C03670=1113.021,-63.508,-48.459,179.722,5.253,148.994
C03671=1113.016,-63.258,-48.470,179.723,5.257,148.995
C03672=1113.010,-63.008,-48.481,179.723,5.262,148.995
C03673=1113.006,-62.759,-48.493,179.724,5.268,148.997
C03674=1113.001,-62.509,-48.504,179.724,5.273,148.998
C03675=1112.995,-62.259,-48.516,179.724,5.278,148.998
C03676=1112.990,-62.010,-48.526,179.725,5.283,148.999
C03677=1112.985,-61.760,-48.537,179.725,5.288,149.001
C03678=1112.980,-61.510,-48.549,179.726,5.293,149.001
C03679=1112.975,-61.260,-48.560,179.726,5.298,149.002
C03680=1112.969,-61.011,-48.572,179.727,5.303,149.003
C03681=1112.964,-60.761,-48.583,179.727,5.308,149.004
C03682=1112.959,-60.511,-48.594,179.727,5.313,149.005
C03683=1112.954,-60.261,-48.606,179.728,5.319,149.006
C03684=1112.949,-60.013,-48.617,179.729,5.324,149.007
C03685=1112.944,-59.798,-48.627,179.728,5.327,149.008
C03686=1112.940,-59.583,-48.637,179.728,5.331,149.009
C03687=1112.936,-59.368,-48.647,179.728,5.335,149.010
C03688=1112.930,-59.153,-48.656,179.728,5.339,149.011
C03689=1112.926,-58.938,-48.666,179.728,5.343,149.012
C03690=1112.922,-58.723,-48.676,179.728,5.348,149.013
C03691=1112.917,-58.509,-48.686,179.728,5.352,149.014
C03692=1112.913,-58.294,-48.696,179.728,5.356,149.015
C03693=1112.907,-58.044,-48.707,179.727,5.360,149.016
C03694=1112.902,-57.795,-48.718,179.727,5.365,149.017
C03695=1112.897,-57.545,-48.730,179.728,5.370,149.018
C03696=1112.892,-57.295,-48.742,179.727,5.374,149.019
C03697=1112.887,-57.045,-48.753,179.727,5.379,149.020
C03698=1112.882,-56.796,-48.765,179.727,5.384,149.021
C03699=1112.876,-56.546,-48.776,179.727,5.388,149.022
C03700=1112.871,-56.297,-48.788,179.727,5.393,149.023
C03701=1112.866,-56.047,-48.799,179.726,5.397,149.024
C03702=1112.861,-55.797,-48.811,179.726,5.403,149.025
C03703=1112.856,-55.547,-48.823,179.727,5.407,149.026
C03704=1112.851,-55.298,-48.834,179.726,5.412,149.027
C03705=1112.845,-55.048,-48.845,179.726,5.417,149.028
C03706=1112.840,-54.799,-48.857,179.726,5.421,149.029
C03707=1112.835,-54.549,-48.869,179.726,5.426,149.031
C03708=1112.829,-54.299,-48.881,179.726,5.431,149.032
C03709=1112.825,-54.049,-48.892,179.725,5.435,149.033
C03710=1112.819,-53.799,-48.904,179.725,5.440,149.034
C03711=1112.814,-53.549,-48.916,179.725,5.445,149.035
C03712=1112.809,-53.301,-48.927,179.725,5.449,149.036
C03713=1112.803,-53.051,-48.938,179.725,5.454,149.037
C03714=1112.799,-52.801,-48.950,179.724,5.459,149.038
C03715=1112.793,-52.551,-48.962,179.725,5.463,149.039
C03716=1112.788,-52.302,-48.974,179.725,5.468,149.040
C03717=1112.783,-52.052,-48.985,179.724,5.473,149.041
C03718=1112.778,-51.802,-48.997,179.724,5.478,149.042
C03719=1112.772,-51.552,-49.009,179.724,5.483,149.043
C03720=1112.767,-51.303,-49.020,179.724,5.487,149.045
C03721=1112.762,-51.053,-49.032,179.724,5.492,149.046
C03722=1112.756,-50.803,-49.044,179.723,5.496,149.047
C03723=1112.752,-50.554,-49.055,179.723,5.501,149.048
C03724=1112.746,-50.305,-49.068,179.724,5.506,149.049
C03725=1112.741,-50.055,-49.080,179.723,5.510,149.050
C03726=1112.736,-49.805,-49.091,179.723,5.515,149.051
C03727=1112.731,-49.555,-49.103,179.723,5.521,149.052
C03728=1112.725,-49.305,-49.115,179.723,5.524,149.053
C03729=1112.721,-49.056,-49.127,179.723,5.530,149.054
C03730=1112.716,-48.806,-49.139,179.722,5.534,149.055
C03731=1112.710,-48.556,-49.151,179.722,5.539,149.056
C03732=1112.705,-48.307,-49.161,179.722,5.544,149.057
C03733=1112.699,-48.057,-49.173,179.722,5.548,149.059
C03734=1112.694,-47.808,-49.186,179.722,5.553,149.060
C03735=1112.689,-47.558,-49.198,179.721,5.557,149.061
C03736=1112.684,-47.308,-49.209,179.721,5.562,149.062
C03737=1112.679,-47.059,-49.221,179.721,5.567,149.063
C03738=1112.674,-46.809,-49.234,179.721,5.571,149.064
C03739=1112.668,-46.559,-49.245,179.721,5.577,149.065
C03740=1112.664,-46.310,-49.257,179.721,5.582,149.066
C03741=1112.659,-46.095,-49.268,179.721,5.586,149.067
C03742=1112.654,-45.880,-49.278,179.721,5.590,149.068
C03743=1112.650,-45.665,-49.288,179.720,5.594,149.069
C03744=1112.646,-45.450,-49.298,179.720,5.597,149.070
C03745=1112.642,-45.236,-49.309,179.720,5.601,149.071
C03746=1112.637,-45.021,-49.319,179.720,5.605,149.072
C03747=1112.632,-44.807,-49.329,179.720,5.609,149.073
C03748=1112.628,-44.593,-49.340,179.720,5.613,149.074
C03749=1112.622,-44.343,-49.352,179.719,5.618,149.075
C03750=1112.617,-44.093,-49.364,179.719,5.623,149.076
C03751=1112.612,-43.843,-49.376,179.719,5.627,149.077
C03752=1112.607,-43.594,-49.387,179.719,5.633,149.078
C03753=1112.602,-43.344,-49.399,179.718,5.637,149.079
C03754=1112.596,-43.095,-49.412,179.718,5.642,149.080
C03755=1112.591,-42.845,-49.424,179.719,5.647,149.081
C03756=1112.587,-42.595,-49.437,179.719,5.652,149.082
C03757=1112.582,-42.345,-49.448,179.720,5.657,149.083
C03758=1112.576,-42.095,-49.460,179.721,5.663,149.084
C03759=1112.571,-41.846,-49.473,179.722,5.667,149.085
C03760=1112.566,-41.596,-49.484,179.723,5.673,149.086
C03761=1112.561,-41.347,-49.497,179.723,5.678,149.087
C03762=1112.555,-41.097,-49.509,179.724,5.683,149.087
C03763=1112.550,-40.847,-49.522,179.725,5.688,149.088
C03764=1112.545,-40.597,-49.533,179.726,5.693,149.089
C03765=1112.540,-40.348,-49.546,179.726,5.698,149.090
C03766=1112.534,-40.098,-49.558,179.727,5.703,149.091
C03767=1112.530,-39.849,-49.570,179.728,5.708,149.092
C03768=1112.524,-39.599,-49.582,179.729,5.713,149.093
C03769=1112.519,-39.350,-49.594,179.729,5.718,149.094
C03770=1112.514,-39.100,-49.606,179.730,5.723,149.094
C03771=1112.509,-38.851,-49.619,179.731,5.728,149.095
C03772=1112.504,-38.600,-49.631,179.732,5.732,149.096
C03773=1112.499,-38.351,-49.644,179.732,5.737,149.097
C03774=1112.494,-38.101,-49.656,179.732,5.742,149.098
C03775=1112.488,-37.851,-49.668,179.733,5.746,149.099
C03776=1112.483,-37.602,-49.681,179.734,5.752,149.100
C03777=1112.478,-37.352,-49.693,179.735,5.756,149.100
C03778=1112.473,-37.103,-49.705,179.735,5.761,149.101
C03779=1112.467,-36.853,-49.718,179.736,5.766,149.102
C03780=1112.462,-36.604,-49.730,179.736,5.771,149.103
C03781=1112.457,-36.353,-49.743,179.737,5.775,149.104
C03782=1112.452,-36.104,-49.755,179.738,5.780,149.105
C03783=1112.447,-35.854,-49.767,179.738,5.784,149.106
C03784=1112.442,-35.605,-49.780,179.738,5.788,149.106
C03785=1112.437,-35.356,-49.792,179.738,5.793,149.107
C03786=1112.430,-35.105,-49.805,179.739,5.797,149.108
C03787=1112.426,-34.855,-49.818,179.740,5.802,149.109
C03788=1112.421,-34.606,-49.830,179.740,5.807,149.110
C03789=1112.416,-34.357,-49.843,179.741,5.812,149.111
C03790=1112.410,-34.107,-49.855,179.740,5.816,149.112
C03791=1112.405,-33.857,-49.868,179.741,5.820,149.113
C03792=1112.401,-33.607,-49.881,179.742,5.825,149.113
C03793=1112.396,-33.358,-49.893,179.742,5.829,149.114
C03794=1112.390,-33.108,-49.905,179.742,5.833,149.115
C03795=1112.385,-32.859,-49.918,179.743,5.838,149.116
C03796=1112.380,-32.610,-49.930,179.743,5.843,149.117
C03797=1112.375,-32.395,-49.942,179.743,5.846,149.118
C03798=1112.371,-32.179,-49.952,179.743,5.850,149.118
C03799=1112.367,-31.965,-49.963,179.744,5.854,149.119
C03800=1112.363,-31.751,-49.974,179.743,5.858,149.120
C03801=1112.358,-31.536,-49.985,179.744,5.861,149.121
C03802=1112.353,-31.321,-49.995,179.744,5.865,149.121
C03803=1112.349,-31.107,-50.007,179.744,5.869,149.122
C03804=1112.345,-30.892,-50.017,179.744,5.872,149.123
C03805=1112.339,-30.643,-50.031,179.745,5.877,149.124
C03806=1112.334,-30.393,-50.043,179.745,5.881,149.125
C03807=1112.329,-30.143,-50.056,179.745,5.886,149.126
C03808=1112.324,-29.894,-50.069,179.745,5.890,149.127
C03809=1112.319,-29.644,-50.081,179.745,5.895,149.128
C03810=1112.314,-29.394,-50.094,179.745,5.899,149.129
C03811=1112.308,-29.145,-50.107,179.745,5.903,149.130
C03812=1112.303,-28.895,-50.119,179.745,5.907,149.130
C03813=1112.298,-28.646,-50.132,179.745,5.912,149.132
C03814=1112.293,-28.396,-50.145,179.745,5.916,149.133
C03815=1112.288,-28.147,-50.157,179.745,5.920,149.133
C03816=1112.282,-27.897,-50.171,179.745,5.925,149.134
C03817=1112.278,-27.647,-50.184,179.745,5.929,149.135
C03818=1112.273,-27.398,-50.196,179.745,5.933,149.136
C03819=1112.268,-27.148,-50.209,179.745,5.939,149.137
C03820=1112.262,-26.899,-50.222,179.744,5.942,149.138
C03821=1112.257,-26.649,-50.235,179.744,5.946,149.139
C03822=1112.252,-26.399,-50.248,179.744,5.952,149.140
C03823=1112.247,-26.150,-50.260,179.744,5.956,149.142
C03824=1112.242,-25.900,-50.274,179.744,5.960,149.142
C03825=1112.237,-25.650,-50.286,179.744,5.965,149.144
C03826=1112.232,-25.401,-50.299,179.744,5.970,149.145
C03827=1112.227,-25.151,-50.312,179.744,5.974,149.145
C03828=1112.221,-24.901,-50.325,179.745,5.979,149.146
C03829=1112.216,-24.652,-50.338,179.745,5.984,149.147
C03830=1112.211,-24.402,-50.351,179.746,5.989,149.148
C03831=1112.206,-24.152,-50.364,179.746,5.993,149.149
C03832=1112.200,-23.903,-50.377,179.747,5.998,149.150
C03833=1112.196,-23.653,-50.389,179.747,6.003,149.151
C03834=1112.190,-23.403,-50.403,179.748,6.007,149.152
C03835=1112.185,-23.154,-50.415,179.748,6.012,149.153
C03836=1112.180,-22.904,-50.428,179.749,6.017,149.154
C03837=1112.175,-22.655,-50.441,179.749,6.022,149.154
C03838=1112.170,-22.406,-50.455,179.750,6.026,149.155
C03839=1112.165,-22.156,-50.468,179.750,6.031,149.156
C03840=1112.159,-21.906,-50.481,179.751,6.036,149.157
C03841=1112.154,-21.657,-50.494,179.751,6.041,149.158
C03842=1112.149,-21.407,-50.507,179.752,6.045,149.159
C03843=1112.144,-21.157,-50.520,179.752,6.050,149.160
C03844=1112.140,-20.908,-50.533,179.753,6.055,149.161
C03845=1112.134,-20.658,-50.547,179.753,6.059,149.162
C03846=1112.129,-20.409,-50.559,179.754,6.064,149.163
C03847=1112.123,-20.159,-50.573,179.754,6.069,149.163
C03848=1112.118,-19.909,-50.585,179.754,6.073,149.164
C03849=1112.114,-19.660,-50.599,179.754,6.078,149.165
C03850=1112.108,-19.410,-50.612,179.755,6.082,149.166
C03851=1112.104,-19.160,-50.625,179.755,6.087,149.167
C03852=1112.098,-18.911,-50.638,179.756,6.092,149.168
C03853=1112.093,-18.697,-50.650,179.757,6.096,149.169
C03854=1112.089,-18.482,-50.661,179.757,6.100,149.169
C03855=1112.085,-18.267,-50.673,179.757,6.104,149.170
C03856=1112.080,-18.053,-50.684,179.758,6.108,149.171
C03857=1112.076,-17.838,-50.695,179.758,6.111,149.171
C03858=1112.072,-17.624,-50.706,179.759,6.116,149.172
C03859=1112.068,-17.409,-50.719,179.759,6.120,149.173
C03860=1112.063,-17.195,-50.730,179.760,6.123,149.174
C03861=1112.058,-16.945,-50.742,179.760,6.128,149.175
C03862=1112.053,-16.696,-50.757,179.761,6.133,149.176
C03863=1112.048,-16.446,-50.769,179.761,6.137,149.176
C03864=1112.042,-16.196,-50.783,179.762,6.142,149.177
C03865=1112.038,-15.947,-50.796,179.763,6.147,149.178
C03866=1112.032,-15.697,-50.810,179.763,6.151,149.179
C03867=1112.027,-15.448,-50.822,179.764,6.156,149.180
C03868=1112.022,-15.198,-50.837,179.764,6.161,149.181
C03869=1112.016,-14.948,-50.850,179.765,6.165,149.182
C03870=1112.012,-14.699,-50.864,179.765,6.170,149.182
C03871=1112.006,-14.449,-50.877,179.766,6.175,149.183
C03872=1112.002,-14.199,-50.890,179.767,6.179,149.184
C03873=1111.996,-13.950,-50.904,179.766,6.183,149.185
C03874=1111.992,-13.700,-50.917,179.767,6.188,149.186
C03875=1111.986,-13.451,-50.930,179.767,6.193,149.187
C03876=1111.981,-13.201,-50.944,179.768,6.197,149.187
C03877=1111.976,-12.952,-50.957,179.769,6.202,149.188
C03878=1111.971,-12.702,-50.971,179.769,6.206,149.189
C03879=1111.966,-12.453,-50.984,179.770,6.211,149.190
C03880=1111.961,-12.203,-50.998,179.771,6.215,149.191
C03881=1111.956,-11.953,-51.012,179.771,6.220,149.192
C03882=1111.951,-11.704,-51.025,179.772,6.225,149.193
C03883=1111.946,-11.454,-51.039,179.772,6.230,149.193
C03884=1111.940,-11.204,-51.052,179.773,6.233,149.194
C03885=1111.936,-10.955,-51.066,179.773,6.238,149.195
C03886=1111.930,-10.706,-51.080,179.774,6.243,149.196
C03887=1111.925,-10.456,-51.093,179.774,6.247,149.197
C03888=1111.921,-10.206,-51.107,179.775,6.252,149.197
C03889=1111.915,-9.957,-51.120,179.776,6.256,149.198
C03890=1111.910,-9.707,-51.134,179.776,6.261,149.199
C03891=1111.905,-9.458,-51.148,179.777,6.266,149.200
C03892=1111.900,-9.208,-51.161,179.778,6.270,149.201
C03893=1111.895,-8.958,-51.176,179.778,6.275,149.202
C03894=1111.890,-8.709,-51.188,179.778,6.279,149.203
C03895=1111.885,-8.459,-51.202,179.779,6.284,149.203
C03896=1111.880,-8.209,-51.217,179.780,6.288,149.204
C03897=1111.874,-7.960,-51.230,179.780,6.293,149.205
C03898=1111.870,-7.710,-51.244,179.781,6.297,149.206
C03899=1111.864,-7.461,-51.258,179.782,6.302,149.207
C03900=1111.859,-7.212,-51.272,179.782,6.306,149.207
C03901=1111.854,-6.961,-51.285,179.783,6.311,149.208
C03902=1111.849,-6.713,-51.299,179.783,6.316,149.209
C03903=1111.844,-6.463,-51.313,179.784,6.320,149.210
C03904=1111.839,-6.213,-51.327,179.784,6.324,149.211
C03905=1111.833,-5.964,-51.340,179.785,6.329,149.212
C03906=1111.829,-5.714,-51.354,179.786,6.333,149.212
C03907=1111.824,-5.464,-51.368,179.786,6.338,149.213
C03908=1111.818,-5.215,-51.382,179.787,6.343,149.214
C03909=1111.814,-5.000,-51.394,179.787,6.346,149.215
C03910=1111.810,-4.786,-51.406,179.788,6.350,149.215
C03911=1111.806,-4.571,-51.418,179.788,6.354,149.216
C03912=1111.801,-4.357,-51.430,179.788,6.358,149.217
C03913=1111.797,-4.143,-51.442,179.789,6.362,149.218
C03914=1111.793,-3.928,-51.453,179.790,6.366,149.218
C03915=1111.788,-3.714,-51.466,179.790,6.369,149.219
C03916=1111.784,-3.499,-51.478,179.791,6.374,149.220
C03917=1111.779,-3.250,-51.492,179.792,6.378,149.221
C03918=1111.774,-3.000,-51.505,179.792,6.383,149.222
C03919=1111.769,-2.750,-51.520,179.793,6.387,149.222
C03920=1111.763,-2.501,-51.534,179.793,6.391,149.223
C03921=1111.758,-2.252,-51.548,179.794,6.396,149.224
C03922=1111.753,-2.002,-51.562,179.794,6.401,149.225
C03923=1111.748,-1.752,-51.576,179.795,6.405,149.226
C03924=1111.743,-1.503,-51.590,179.796,6.410,149.226
C03925=1111.738,-1.253,-51.605,179.796,6.415,149.227
C03926=1111.733,-1.004,-51.618,179.797,6.419,149.228
C03927=1111.729,-0.754,-51.633,179.798,6.424,149.229
C03928=1111.723,-0.505,-51.646,179.798,6.428,149.230
C03929=1111.718,-0.256,-51.661,179.798,6.432,149.231
C03930=1111.713,-0.006,-51.675,179.799,6.437,149.231
C03931=1111.708,0.244,-51.689,179.800,6.441,149.232
C03932=1111.702,0.493,-51.702,179.800,6.446,149.233
C03933=1111.697,0.743,-51.717,179.801,6.450,149.234
C03934=1111.692,0.993,-51.731,179.802,6.455,149.235
C03935=1111.688,1.242,-51.746,179.802,6.460,149.236
C03936=1111.683,1.492,-51.760,179.803,6.464,149.236
C03937=1111.677,1.741,-51.774,179.804,6.469,149.237
C03938=1111.672,1.990,-51.788,179.804,6.474,149.238
C03939=1111.667,2.240,-51.803,179.804,6.477,149.239
C03940=1111.662,2.490,-51.817,179.805,6.482,149.240
C03941=1111.657,2.740,-51.831,179.806,6.486,149.240
C03942=1111.652,2.989,-51.845,179.806,6.491,149.241
C03943=1111.647,3.238,-51.860,179.807,6.496,149.242
C03944=1111.642,3.488,-51.874,179.807,6.501,149.243
C03945=1111.637,3.738,-51.888,179.808,6.505,149.244
C03946=1111.632,3.987,-51.902,179.809,6.510,149.245
C03947=1111.627,4.237,-51.917,179.810,6.514,149.245
C03948=1111.622,4.486,-51.932,179.810,6.519,149.246
C03949=1111.617,4.735,-51.946,179.811,6.523,149.247
C03950=1111.611,4.985,-51.960,179.812,6.528,149.248
C03951=1111.606,5.235,-51.975,179.812,6.533,149.249
C03952=1111.601,5.485,-51.989,179.812,6.537,149.250
C03953=1111.596,5.734,-52.003,179.813,6.541,149.251
C03954=1111.592,5.983,-52.018,179.814,6.546,149.251
C03955=1111.587,6.233,-52.033,179.814,6.551,149.252
C03956=1111.581,6.482,-52.046,179.815,6.555,149.253
C03957=1111.576,6.732,-52.061,179.815,6.560,149.254
C03958=1111.572,6.981,-52.076,179.816,6.565,149.255
C03959=1111.566,7.231,-52.091,179.817,6.569,149.255
C03960=1111.561,7.481,-52.105,179.817,6.574,149.256
C03961=1111.556,7.730,-52.119,179.818,6.578,149.257
C03962=1111.551,7.979,-52.134,179.818,6.583,149.258
C03963=1111.546,8.229,-52.148,179.819,6.588,149.259
C03964=1111.541,8.479,-52.163,179.820,6.593,149.260
C03965=1111.536,8.693,-52.175,179.820,6.596,149.261
C03966=1111.532,8.908,-52.188,179.820,6.600,149.261
C03967=1111.528,9.121,-52.200,179.821,6.604,149.262
C03968=1111.524,9.336,-52.213,179.821,6.608,149.263
C03969=1111.520,9.551,-52.226,179.822,6.611,149.263
C03970=1111.515,9.765,-52.238,179.822,6.616,149.264
C03971=1111.511,9.980,-52.251,179.823,6.620,149.265
C03972=1111.506,10.193,-52.263,179.823,6.623,149.266
C03973=1111.501,10.443,-52.278,179.824,6.628,149.267
C03974=1111.496,10.693,-52.293,179.824,6.633,149.267
C03975=1111.491,10.942,-52.307,179.825,6.637,149.268
C03976=1111.486,11.191,-52.322,179.826,6.642,149.269
C03977=1111.481,11.441,-52.336,179.826,6.646,149.270
C03978=1111.476,11.691,-52.352,179.826,6.650,149.271
C03979=1111.471,11.940,-52.366,179.827,6.655,149.272
C03980=1111.466,12.189,-52.381,179.827,6.660,149.272
C03981=1111.461,12.439,-52.395,179.828,6.664,149.273
C03982=1111.456,12.689,-52.410,179.829,6.669,149.274
C03983=1111.451,12.938,-52.425,179.830,6.673,149.275
C03984=1111.446,13.188,-52.440,179.829,6.677,149.276
C03985=1111.441,13.437,-52.455,179.830,6.682,149.276
C03986=1111.436,13.687,-52.469,179.831,6.686,149.277
C03987=1111.431,13.936,-52.484,179.832,6.691,149.278
C03988=1111.425,14.186,-52.499,179.833,6.695,149.279
C03989=1111.421,14.435,-52.514,179.833,6.700,149.280
C03990=1111.416,14.685,-52.529,179.833,6.704,149.281
C03991=1111.410,14.934,-52.544,179.834,6.709,149.282
C03992=1111.405,15.184,-52.558,179.835,6.713,149.282
C03993=1111.401,15.433,-52.573,179.835,6.718,149.283
C03994=1111.395,15.682,-52.589,179.836,6.722,149.284
C03995=1111.390,15.932,-52.603,179.837,6.727,149.285
C03996=1111.386,16.181,-52.618,179.837,6.731,149.285
C03997=1111.380,16.431,-52.633,179.838,6.735,149.286
C03998=1111.376,16.681,-52.649,179.838,6.740,149.287
C03999=1111.371,16.930,-52.664,179.839,6.744,149.288
C04000=1111.366,17.180,-52.678,179.840,6.749,149.289
C04001=1111.361,17.429,-52.693,179.841,6.753,149.289
C04002=1111.355,17.679,-52.708,179.841,6.757,149.290
C04003=1111.351,17.928,-52.723,179.842,6.762,149.291
C04004=1111.345,18.178,-52.739,179.843,6.766,149.292
C04005=1111.340,18.428,-52.753,179.843,6.771,149.293
C04006=1111.336,18.677,-52.768,179.844,6.775,149.293
C04007=1111.330,18.926,-52.784,179.844,6.779,149.294
C04008=1111.326,19.175,-52.799,179.845,6.784,149.295
C04009=1111.320,19.425,-52.814,179.846,6.788,149.296
C04010=1111.316,19.675,-52.829,179.846,6.793,149.296
C04011=1111.310,19.924,-52.844,179.847,6.797,149.297
C04012=1111.306,20.174,-52.859,179.848,6.802,149.298
C04013=1111.300,20.423,-52.874,179.848,6.805,149.299
C04014=1111.296,20.673,-52.889,179.849,6.809,149.299
C04015=1111.290,20.922,-52.905,179.850,6.814,149.300
C04016=1111.285,21.172,-52.919,179.851,6.818,149.301
C04017=1111.280,21.422,-52.935,179.852,6.823,149.302
C04018=1111.276,21.671,-52.950,179.852,6.827,149.302
C04019=1111.270,21.920,-52.966,179.853,6.831,149.303
C04020=1111.266,22.169,-52.981,179.854,6.836,149.304
C04021=1111.261,22.384,-52.994,179.854,6.839,149.305
C04022=1111.256,22.598,-53.007,179.855,6.844,149.305
C04023=1111.252,22.813,-53.019,179.856,6.847,149.306
C04024=1111.248,23.027,-53.033,179.856,6.851,149.307
C04025=1111.244,23.241,-53.046,179.856,6.854,149.307
C04026=1111.239,23.455,-53.059,179.857,6.858,149.308
C04027=1111.235,23.669,-53.073,179.858,6.862,149.308
C04028=1111.231,23.883,-53.086,179.859,6.865,149.309
C04029=1111.226,24.133,-53.101,179.859,6.870,149.310
C04030=1111.220,24.383,-53.116,179.860,6.874,149.311
C04031=1111.216,24.633,-53.132,179.861,6.878,149.311
C04032=1111.211,24.882,-53.147,179.861,6.882,149.312
C04033=1111.206,25.131,-53.162,179.863,6.887,149.313
C04034=1111.201,25.381,-53.178,179.864,6.891,149.313
C04035=1111.195,25.630,-53.193,179.864,6.896,149.314
C04036=1111.191,25.880,-53.209,179.865,6.900,149.315
C04037=1111.186,26.129,-53.224,179.866,6.903,149.316
C04038=1111.181,26.378,-53.239,179.866,6.908,149.316
C04039=1111.176,26.628,-53.255,179.867,6.912,149.317
C04040=1111.171,26.878,-53.271,179.868,6.917,149.318
C04041=1111.167,27.127,-53.286,179.869,6.921,149.318
C04042=1111.161,27.376,-53.301,179.869,6.925,149.319
C04043=1111.156,27.626,-53.317,179.870,6.929,149.320
C04044=1111.151,27.876,-53.333,179.871,6.934,149.321
C04045=1111.146,28.125,-53.348,179.872,6.938,149.321
C04046=1111.141,28.374,-53.363,179.874,6.942,149.322
C04047=1111.136,28.624,-53.379,179.874,6.946,149.323
C04048=1111.132,28.873,-53.394,179.875,6.950,149.323
C04049=1111.126,29.123,-53.410,179.876,6.955,149.324
C04050=1111.121,29.372,-53.426,179.877,6.959,149.325
C04051=1111.116,29.621,-53.441,179.877,6.963,149.325
C04052=1111.111,29.871,-53.457,179.878,6.967,149.326
C04053=1111.106,30.120,-53.473,179.879,6.972,149.327
C04054=1111.101,30.370,-53.488,179.880,6.976,149.328
C04055=1111.097,30.619,-53.504,179.881,6.980,149.328
C04056=1111.091,30.869,-53.519,179.881,6.984,149.329
C04057=1111.086,31.118,-53.535,179.882,6.988,149.330
C04058=1111.081,31.368,-53.551,179.883,6.993,149.330
C04059=1111.076,31.618,-53.567,179.884,6.997,149.331
C04060=1111.072,31.866,-53.582,179.885,7.001,149.332
C04061=1111.067,32.116,-53.598,179.886,7.005,149.332
C04062=1111.061,32.366,-53.614,179.887,7.009,149.333
C04063=1111.056,32.615,-53.629,179.888,7.014,149.334
C04064=1111.051,32.865,-53.645,179.889,7.018,149.334
C04065=1111.047,33.114,-53.661,179.890,7.022,149.335
C04066=1111.041,33.363,-53.677,179.890,7.026,149.336
C04067=1111.037,33.613,-53.693,179.891,7.030,149.336
C04068=1111.031,33.863,-53.708,179.892,7.034,149.337
C04069=1111.026,34.111,-53.724,179.893,7.039,149.338
C04070=1111.021,34.362,-53.740,179.894,7.043,149.338
C04071=1111.016,34.611,-53.756,179.894,7.047,149.339
C04072=1111.012,34.860,-53.772,179.896,7.051,149.340
C04073=1111.007,35.109,-53.788,179.897,7.055,149.340
C04074=1111.002,35.359,-53.803,179.898,7.060,149.341
C04075=1110.997,35.608,-53.820,179.898,7.063,149.342
C04076=1110.992,35.858,-53.836,179.899,7.068,149.342
C04077=1110.987,36.072,-53.849,179.900,7.071,149.343
C04078=1110.983,36.286,-53.863,179.901,7.075,149.344
C04079=1110.979,36.501,-53.877,179.902,7.078,149.344
C04080=1110.974,36.715,-53.890,179.903,7.082,149.345
C04081=1110.970,36.929,-53.904,179.904,7.086,149.345
C04082=1110.966,37.144,-53.918,179.905,7.089,149.346
C04083=1110.962,37.357,-53.932,179.905,7.093,149.346
C04084=1110.957,37.571,-53.946,179.906,7.096,149.347
C04085=1110.953,37.821,-53.961,179.907,7.100,149.347
C04086=1110.948,38.070,-53.977,179.908,7.104,149.348
C04087=1110.943,38.320,-53.993,179.909,7.109,149.349
C04088=1110.938,38.569,-54.009,179.910,7.112,149.349
C04089=1110.933,38.819,-54.025,179.911,7.116,149.350
C04090=1110.928,39.068,-54.041,179.912,7.121,149.351
C04091=1110.923,39.317,-54.058,179.913,7.125,149.351
C04092=1110.918,39.567,-54.073,179.914,7.129,149.352
C04093=1110.913,39.816,-54.090,179.915,7.133,149.352
C04094=1110.908,40.066,-54.105,179.916,7.137,149.353
C04095=1110.903,40.315,-54.122,179.917,7.141,149.354
C04096=1110.898,40.565,-54.138,179.918,7.145,149.354
C04097=1110.892,40.814,-54.155,179.919,7.150,149.355
C04098=1110.888,41.064,-54.171,179.919,7.153,149.356
C04099=1110.883,41.313,-54.187,179.921,7.158,149.356
C04100=1110.878,41.562,-54.204,179.922,7.161,149.357
C04101=1110.873,41.812,-54.219,179.923,7.166,149.357
C04102=1110.868,42.061,-54.236,179.924,7.169,149.358
C04103=1110.863,42.310,-54.251,179.925,7.174,149.359
C04104=1110.858,42.560,-54.268,179.926,7.178,149.359
C04105=1110.854,42.810,-54.284,179.927,7.182,149.360
C04106=1110.848,43.059,-54.300,179.928,7.186,149.361
C04107=1110.844,43.308,-54.317,179.929,7.190,149.361
C04108=1110.839,43.558,-54.333,179.930,7.194,149.362
C04109=1110.834,43.807,-54.349,179.931,7.198,149.362
C04110=1110.828,44.056,-54.366,179.932,7.203,149.363
C04111=1110.824,44.306,-54.382,179.934,7.206,149.364
C04112=1110.818,44.555,-54.398,179.934,7.210,149.364
C04113=1110.814,44.805,-54.415,179.935,7.214,149.365
C04114=1110.809,45.055,-54.431,179.936,7.219,149.366
C04115=1110.804,45.304,-54.447,179.937,7.223,149.366
C04116=1110.800,45.553,-54.464,179.939,7.227,149.367
C04117=1110.794,45.802,-54.481,179.939,7.230,149.367
C04118=1110.789,46.052,-54.497,179.940,7.235,149.368
C04119=1110.784,46.301,-54.513,179.942,7.239,149.369
C04120=1110.779,46.550,-54.530,179.943,7.243,149.369
C04121=1110.775,46.800,-54.547,179.944,7.247,149.370
C04122=1110.769,47.050,-54.563,179.945,7.251,149.370
C04123=1110.764,47.299,-54.579,179.946,7.255,149.371
C04124=1110.760,47.549,-54.596,179.947,7.259,149.371
C04125=1110.755,47.797,-54.612,179.948,7.263,149.372
C04126=1110.750,48.047,-54.629,179.949,7.267,149.373
C04127=1110.745,48.296,-54.646,179.950,7.271,149.373
C04128=1110.740,48.546,-54.662,179.951,7.275,149.374
C04129=1110.735,48.796,-54.679,179.952,7.279,149.374
C04130=1110.730,49.044,-54.695,179.954,7.283,149.375
C04131=1110.725,49.294,-54.712,179.955,7.287,149.376
C04132=1110.720,49.544,-54.729,179.956,7.291,149.376
C04133=1110.716,49.758,-54.742,179.957,7.295,149.377
C04134=1110.712,49.972,-54.757,179.958,7.298,149.377
C04135=1110.707,50.186,-54.772,179.959,7.301,149.378
C04136=1110.703,50.400,-54.786,179.959,7.305,149.378
C04137=1110.699,50.614,-54.800,179.961,7.308,149.379
C04138=1110.695,50.828,-54.814,179.962,7.312,149.379
C04139=1110.690,51.042,-54.829,179.962,7.315,149.380
C04140=1110.686,51.256,-54.843,179.963,7.318,149.380
C04141=1110.682,51.505,-54.860,179.964,7.323,149.381
C04142=1110.676,51.755,-54.877,179.966,7.326,149.381
C04143=1110.671,52.004,-54.893,179.967,7.331,149.382
C04144=1110.667,52.253,-54.910,179.969,7.335,149.382
C04145=1110.662,52.503,-54.927,179.970,7.339,149.383
C04146=1110.657,52.753,-54.944,179.970,7.342,149.384
C04147=1110.652,53.001,-54.960,179.972,7.346,149.384
C04148=1110.647,53.251,-54.978,179.973,7.351,149.385
C04149=1110.642,53.501,-54.994,179.974,7.355,149.385
C04150=1110.637,53.750,-55.011,179.975,7.359,149.386
C04151=1110.632,53.999,-55.028,179.976,7.362,149.386
C04152=1110.628,54.249,-55.045,179.978,7.366,149.387
C04153=1110.622,54.498,-55.062,179.979,7.371,149.387
C04154=1110.617,54.747,-55.078,179.980,7.375,149.388
C04155=1110.612,54.997,-55.095,179.981,7.379,149.389
C04156=1110.608,55.247,-55.112,179.983,7.383,149.389
C04157=1110.603,55.496,-55.130,179.983,7.386,149.390
C04158=1110.598,55.745,-55.146,179.985,7.390,149.390
C04159=1110.592,55.994,-55.164,179.986,7.394,149.391
C04160=1110.588,56.244,-55.180,179.987,7.399,149.391
C04161=1110.583,56.494,-55.197,179.989,7.403,149.392
C04162=1110.578,56.743,-55.214,179.989,7.406,149.392
C04163=1110.573,56.992,-55.230,179.991,7.410,149.393
C04164=1110.568,57.241,-55.248,179.992,7.414,149.394
C04165=1110.563,57.491,-55.266,179.993,7.418,149.394
C04166=1110.559,57.740,-55.282,179.994,7.423,149.395
C04167=1110.553,57.990,-55.300,179.996,7.426,149.395
C04168=1110.549,58.238,-55.317,179.996,7.430,149.396
C04169=1110.543,58.488,-55.334,179.998,7.434,149.396
C04170=1110.539,58.738,-55.351,179.999,7.438,149.397
C04171=1110.534,58.987,-55.368,-179.999,7.442,149.397
C04172=1110.529,59.236,-55.385,-179.998,7.446,149.398
C04173=1110.524,59.486,-55.403,-179.997,7.450,149.398
C04174=1110.519,59.735,-55.419,-179.996,7.454,149.399
C04175=1110.514,59.984,-55.437,-179.995,7.458,149.399
C04176=1110.509,60.234,-55.454,-179.994,7.462,149.400
C04177=1110.505,60.483,-55.471,-179.992,7.466,149.400
C04178=1110.500,60.732,-55.489,-179.990,7.470,149.401
C04179=1110.495,60.982,-55.505,-179.989,7.474,149.402
C04180=1110.490,61.232,-55.523,-179.988,7.477,149.402
C04181=1110.484,61.480,-55.540,-179.987,7.482,149.403
C04182=1110.480,61.730,-55.557,-179.986,7.485,149.403
C04183=1110.475,61.979,-55.575,-179.985,7.490,149.404
C04184=1110.471,62.228,-55.592,-179.983,7.494,149.404
C04185=1110.465,62.478,-55.609,-179.982,7.498,149.405
C04186=1110.460,62.727,-55.627,-179.981,7.501,149.405
C04187=1110.456,62.977,-55.643,-179.979,7.505,149.406
C04188=1110.451,63.226,-55.661,-179.978,7.509,149.406
C04189=1110.446,63.440,-55.676,-179.977,7.513,149.407
C04190=1110.442,63.654,-55.691,-179.976,7.516,149.407
C04191=1110.438,63.868,-55.706,-179.975,7.519,149.408
C04192=1110.434,64.082,-55.721,-179.974,7.522,149.408
C04193=1110.429,64.296,-55.736,-179.972,7.526,149.409
C04194=1110.426,64.510,-55.750,-179.971,7.530,149.409
C04195=1110.421,64.725,-55.766,-179.971,7.533,149.409
C04196=1110.418,64.938,-55.781,-179.969,7.537,149.410
C04197=1110.412,65.187,-55.798,-179.968,7.541,149.410
C04198=1110.408,65.437,-55.816,-179.967,7.544,149.411
C04199=1110.402,65.686,-55.833,-179.966,7.548,149.412
C04200=1110.398,65.935,-55.851,-179.964,7.552,149.412
C04201=1110.393,66.185,-55.868,-179.963,7.556,149.412
C04202=1110.388,66.434,-55.886,-179.962,7.560,149.413
C04203=1110.383,66.683,-55.904,-179.960,7.564,149.414
C04204=1110.379,66.933,-55.920,-179.959,7.569,149.414
C04205=1110.374,67.182,-55.938,-179.958,7.572,149.415
C04206=1110.369,67.432,-55.956,-179.956,7.576,149.415
C04207=1110.364,67.681,-55.974,-179.955,7.580,149.416
C04208=1110.359,67.930,-55.992,-179.954,7.584,149.416
C04209=1110.354,68.180,-56.008,-179.952,7.588,149.417
C04210=1110.349,68.429,-56.026,-179.951,7.592,149.417
C04211=1110.344,68.678,-56.044,-179.949,7.596,149.418
C04212=1110.339,68.928,-56.062,-179.948,7.600,149.418
C04213=1110.334,69.177,-56.080,-179.947,7.603,149.419
C04214=1110.329,69.426,-56.098,-179.946,7.607,149.419
C04215=1110.325,69.675,-56.115,-179.944,7.611,149.420
C04216=1110.320,69.925,-56.132,-179.943,7.615,149.420
C04217=1110.315,70.174,-56.150,-179.942,7.619,149.421
C04218=1110.310,70.423,-56.168,-179.940,7.623,149.421
C04219=1110.305,70.672,-56.186,-179.939,7.627,149.422
C04220=1110.300,70.922,-56.203,-179.937,7.631,149.422
C04221=1110.295,71.171,-56.221,-179.936,7.635,149.423
C04222=1110.290,71.420,-56.239,-179.935,7.639,149.423
C04223=1110.286,71.669,-56.257,-179.934,7.643,149.424
C04224=1110.281,71.919,-56.275,-179.932,7.647,149.424
C04225=1110.276,72.168,-56.293,-179.931,7.651,149.425
C04226=1110.272,72.418,-56.310,-179.929,7.655,149.425
C04227=1110.267,72.667,-56.328,-179.928,7.659,149.426
C04228=1110.262,72.917,-56.346,-179.927,7.663,149.426
C04229=1110.257,73.166,-56.364,-179.925,7.667,149.427
C04230=1110.252,73.415,-56.382,-179.924,7.671,149.427
C04231=1110.247,73.664,-56.400,-179.922,7.675,149.428
C04232=1110.242,73.913,-56.418,-179.921,7.678,149.428
C04233=1110.237,74.162,-56.436,-179.920,7.682,149.429
C04234=1110.232,74.412,-56.454,-179.918,7.686,149.429
C04235=1110.228,74.662,-56.472,-179.917,7.690,149.430
C04236=1110.223,74.911,-56.490,-179.916,7.694,149.430
C04237=1110.218,75.160,-56.508,-179.914,7.698,149.431
C04238=1110.213,75.410,-56.526,-179.912,7.702,149.431
C04239=1110.208,75.659,-56.544,-179.911,7.706,149.432
C04240=1110.203,75.908,-56.562,-179.910,7.710,149.432
C04241=1110.198,76.157,-56.580,-179.908,7.714,149.433
C04242=1110.194,76.407,-56.598,-179.907,7.718,149.433
C04243=1110.189,76.656,-56.616,-179.905,7.722,149.434
C04244=1110.184,76.905,-56.634,-179.904,7.726,149.434
C04245=1110.180,77.119,-56.650,-179.904,7.728,149.435
C04246=1110.176,77.333,-56.666,-179.903,7.731,149.435
C04247=1110.171,77.547,-56.681,-179.902,7.735,149.436
C04248=1110.167,77.761,-56.697,-179.901,7.738,149.436
C04249=1110.163,77.974,-56.713,-179.900,7.741,149.436
C04250=1110.159,78.189,-56.728,-179.899,7.744,149.437
C04251=1110.154,78.402,-56.744,-179.898,7.747,149.437
C04252=1110.150,78.617,-56.760,-179.898,7.751,149.438
C04253=1110.146,78.866,-56.778,-179.896,7.755,149.438
C04254=1110.141,79.115,-56.796,-179.896,7.758,149.439
C04255=1110.136,79.364,-56.814,-179.894,7.762,149.440
C04256=1110.131,79.614,-56.832,-179.894,7.766,149.440
C04257=1110.127,79.863,-56.850,-179.892,7.770,149.441
C04258=1110.122,80.112,-56.868,-179.891,7.773,149.441
C04259=1110.116,80.361,-56.887,-179.890,7.777,149.442
C04260=1110.112,80.611,-56.906,-179.889,7.781,149.442
C04261=1110.107,80.860,-56.924,-179.888,7.785,149.443
C04262=1110.102,81.109,-56.942,-179.887,7.788,149.443
C04263=1110.097,81.359,-56.960,-179.886,7.792,149.444
C04264=1110.093,81.608,-56.979,-179.885,7.795,149.444
C04265=1110.088,81.857,-56.997,-179.884,7.800,149.445
C04266=1110.083,82.107,-57.015,-179.883,7.803,149.446
C04267=1110.078,82.356,-57.033,-179.882,7.807,149.446
C04268=1110.074,82.605,-57.052,-179.880,7.811,149.447
C04269=1110.069,82.854,-57.070,-179.880,7.814,149.447
C04270=1110.063,83.104,-57.089,-179.878,7.818,149.448
C04271=1110.058,83.353,-57.107,-179.878,7.822,149.448
C04272=1110.054,83.602,-57.126,-179.876,7.826,149.449
C04273=1110.049,83.851,-57.144,-179.875,7.830,149.449
C04274=1110.044,84.101,-57.162,-179.874,7.833,149.450
C04275=1110.040,84.350,-57.182,-179.873,7.837,149.450
C04276=1110.035,84.599,-57.200,-179.871,7.841,149.451
C04277=1110.030,84.848,-57.218,-179.870,7.844,149.451
C04278=1110.025,85.098,-57.237,-179.869,7.849,149.452
C04279=1110.020,85.347,-57.255,-179.868,7.852,149.452
C04280=1110.015,85.596,-57.273,-179.867,7.856,149.453
C04281=1110.011,85.846,-57.293,-179.866,7.860,149.454
C04282=1110.006,86.095,-57.311,-179.865,7.863,149.454
C04283=1110.001,86.344,-57.329,-179.864,7.867,149.455
C04284=1109.996,86.594,-57.348,-179.862,7.871,149.455
C04285=1109.991,86.843,-57.366,-179.861,7.875,149.456
C04286=1109.986,87.091,-57.385,-179.860,7.879,149.456
C04287=1109.981,87.342,-57.404,-179.858,7.882,149.457
C04288=1109.977,87.590,-57.423,-179.858,7.886,149.457
C04289=1109.972,87.839,-57.441,-179.856,7.890,149.458
C04290=1109.967,88.089,-57.460,-179.855,7.894,149.458
C04291=1109.962,88.338,-57.478,-179.854,7.897,149.459
C04292=1109.957,88.587,-57.498,-179.852,7.901,149.459
C04293=1109.953,88.837,-57.516,-179.851,7.905,149.460
C04294=1109.948,89.085,-57.535,-179.850,7.909,149.460
C04295=1109.943,89.336,-57.554,-179.849,7.912,149.461
C04296=1109.938,89.584,-57.572,-179.847,7.916,149.461
C04297=1109.933,89.834,-57.591,-179.846,7.921,149.462
C04298=1109.929,90.083,-57.610,-179.844,7.924,149.462
C04299=1109.924,90.332,-57.628,-179.843,7.928,149.463
C04300=1109.919,90.582,-57.648,-179.842,7.931,149.463
C04301=1109.915,90.795,-57.663,-179.841,7.935,149.464
C04302=1109.911,91.009,-57.679,-179.840,7.938,149.464
C04303=1109.907,91.223,-57.695,-179.838,7.942,149.464
C04304=1109.902,91.437,-57.712,-179.837,7.945,149.465
C04305=1109.898,91.650,-57.729,-179.836,7.948,149.465
C04306=1109.894,91.865,-57.745,-179.835,7.951,149.466
C04307=1109.890,92.078,-57.760,-179.834,7.955,149.466
C04308=1109.886,92.292,-57.777,-179.833,7.958,149.467
C04309=1109.881,92.541,-57.796,-179.831,7.962,149.467
C04310=1109.877,92.791,-57.814,-179.830,7.965,149.467
C04311=1109.871,93.040,-57.834,-179.829,7.969,149.468
C04312=1109.867,93.289,-57.853,-179.827,7.973,149.468
C04313=1109.862,93.538,-57.871,-179.826,7.977,149.469
C04314=1109.858,93.788,-57.890,-179.824,7.981,149.469
C04315=1109.852,94.037,-57.909,-179.823,7.984,149.470
C04316=1109.848,94.286,-57.929,-179.822,7.988,149.470
C04317=1109.843,94.535,-57.947,-179.820,7.992,149.471
C04318=1109.838,94.785,-57.967,-179.819,7.996,149.471
C04319=1109.833,95.033,-57.985,-179.817,7.999,149.472
C04320=1109.828,95.283,-58.005,-179.816,8.003,149.472
C04321=1109.824,95.532,-58.023,-179.814,8.006,149.472
C04322=1109.819,95.782,-58.043,-179.813,8.011,149.473
C04323=1109.813,96.031,-58.062,-179.812,8.015,149.474
C04324=1109.809,96.280,-58.081,-179.810,8.019,149.474
C04325=1109.804,96.529,-58.100,-179.808,8.022,149.474
C04326=1109.800,96.778,-58.119,-179.807,8.026,149.475
C04327=1109.794,97.027,-58.138,-179.806,8.029,149.475
C04328=1109.790,97.277,-58.158,-179.804,8.033,149.476
C04329=1109.785,97.526,-58.176,-179.803,8.037,149.476
C04330=1109.780,97.775,-58.196,-179.801,8.041,149.477
C04331=1109.775,98.024,-58.215,-179.799,8.045,149.477
C04332=1109.771,98.273,-58.234,-179.798,8.049,149.477
C04333=1109.766,98.523,-58.254,-179.796,8.053,149.478
C04334=1109.761,98.772,-58.273,-179.795,8.055,149.478
C04335=1109.757,99.021,-58.292,-179.793,8.059,149.479
C04336=1109.752,99.270,-58.312,-179.792,8.063,149.479
C04337=1109.747,99.519,-58.331,-179.790,8.067,149.479
C04338=1109.742,99.768,-58.350,-179.788,8.071,149.480
C04339=1109.737,100.018,-58.369,-179.787,8.075,149.480
C04340=1109.732,100.268,-58.389,-179.785,8.079,149.481
C04341=1109.727,100.517,-58.408,-179.784,8.083,149.481
C04342=1109.723,100.765,-58.428,-179.782,8.086,149.481
C04343=1109.718,101.014,-58.447,-179.780,8.090,149.482
C04344=1109.713,101.264,-58.467,-179.779,8.093,149.482
C04345=1109.709,101.513,-58.486,-179.777,8.097,149.483
C04346=1109.704,101.762,-58.505,-179.776,8.101,149.483
C04347=1109.699,102.011,-58.525,-179.774,8.104,149.483
C04348=1109.695,102.261,-58.544,-179.772,8.108,149.484
C04349=1109.689,102.510,-58.564,-179.771,8.112,149.484
C04350=1109.685,102.759,-58.583,-179.769,8.116,149.485
C04351=1109.680,103.009,-58.602,-179.767,8.120,149.485
C04352=1109.675,103.257,-58.622,-179.765,8.123,149.485
C04353=1109.670,103.507,-58.641,-179.764,8.127,149.486
C04354=1109.666,103.756,-58.662,-179.762,8.131,149.486
C04355=1109.661,104.005,-58.681,-179.760,8.135,149.486
C04356=1109.657,104.254,-58.700,-179.758,8.139,149.487
C04357=1109.652,104.468,-58.717,-179.757,8.141,149.487
C04358=1109.648,104.682,-58.734,-179.755,8.145,149.487
C04359=1109.644,104.895,-58.751,-179.754,8.148,149.488
C04360=1109.640,105.109,-58.767,-179.752,8.151,149.488
C04361=1109.636,105.323,-58.784,-179.751,8.155,149.488
C04362=1109.631,105.537,-58.801,-179.749,8.157,149.489
C04363=1109.628,105.750,-58.818,-179.747,8.161,149.489
C04364=1109.623,105.965,-58.835,-179.746,8.164,149.489
C04365=1109.618,106.213,-58.855,-179.744,8.167,149.489
C04366=1109.614,106.462,-58.874,-179.743,8.171,149.490
C04367=1109.609,106.712,-58.894,-179.741,8.175,149.490
C04368=1109.605,106.961,-58.914,-179.739,8.179,149.491
C04369=1109.600,107.209,-58.933,-179.737,8.182,149.491
C04370=1109.595,107.459,-58.953,-179.735,8.186,149.491
C04371=1109.590,107.708,-58.973,-179.733,8.190,149.491
C04372=1109.586,107.958,-58.993,-179.731,8.193,149.492
C04373=1109.580,108.206,-59.012,-179.730,8.197,149.492
C04374=1109.576,108.455,-59.033,-179.728,8.200,149.492
C04375=1109.571,108.705,-59.052,-179.726,8.204,149.493
C04376=1109.566,108.955,-59.072,-179.724,8.208,149.493
C04377=1109.561,109.203,-59.092,-179.722,8.211,149.493
C04378=1109.557,109.452,-59.112,-179.720,8.215,149.494
C04379=1109.552,109.701,-59.132,-179.718,8.219,149.494
C04380=1109.548,109.951,-59.152,-179.716,8.222,149.494
C04381=1109.543,110.200,-59.172,-179.714,8.226,149.494
C04382=1109.538,110.449,-59.191,-179.713,8.230,149.495
C04383=1109.533,110.698,-59.212,-179.710,8.233,149.495
C04384=1109.529,110.947,-59.231,-179.708,8.237,149.495
C04385=1109.524,111.196,-59.252,-179.706,8.240,149.495
C04386=1109.519,111.446,-59.272,-179.705,8.244,149.496
C04387=1109.514,111.695,-59.292,-179.703,8.247,149.496
C04388=1109.509,111.944,-59.312,-179.702,8.251,149.497
C04389=1109.504,112.193,-59.332,-179.700,8.254,149.497
C04390=1109.500,112.442,-59.352,-179.698,8.258,149.497
C04391=1109.495,112.691,-59.372,-179.697,8.261,149.497
C04392=1109.490,112.941,-59.392,-179.695,8.264,149.498
C04393=1109.486,113.190,-59.412,-179.692,8.268,149.498
C04394=1109.482,113.439,-59.433,-179.691,8.272,149.498
C04395=1109.476,113.688,-59.452,-179.689,8.274,149.499
C04396=1109.471,113.937,-59.473,-179.687,8.278,149.499
C04397=1109.467,114.186,-59.493,-179.686,8.282,149.499
C04398=1109.462,114.435,-59.513,-179.684,8.284,149.499
C04399=1109.457,114.684,-59.533,-179.682,8.288,149.500
C04400=1109.452,114.934,-59.553,-179.681,8.292,149.500
C04401=1109.448,115.183,-59.574,-179.679,8.295,149.500
C04402=1109.443,115.432,-59.594,-179.677,8.298,149.501
C04403=1109.439,115.681,-59.615,-179.676,8.302,149.501
C04404=1109.433,115.930,-59.634,-179.673,8.305,149.501
C04405=1109.428,116.179,-59.655,-179.672,8.308,149.501
C04406=1109.424,116.428,-59.675,-179.670,8.312,149.502
C04407=1109.419,116.677,-59.696,-179.668,8.315,149.502
C04408=1109.415,116.927,-59.715,-179.666,8.319,149.502
C04409=1109.409,117.176,-59.736,-179.665,8.322,149.503
C04410=1109.405,117.425,-59.757,-179.663,8.326,149.503
C04411=1109.401,117.674,-59.777,-179.661,8.329,149.503
C04412=1109.396,117.923,-59.797,-179.660,8.332,149.503
C04413=1109.392,118.137,-59.815,-179.658,8.335,149.504
C04414=1109.388,118.350,-59.832,-179.656,8.338,149.504
C04415=1109.383,118.564,-59.850,-179.655,8.341,149.504
C04416=1109.379,118.778,-59.867,-179.654,8.344,149.505
C04417=1109.375,118.991,-59.885,-179.652,8.347,149.505
C04418=1109.372,119.205,-59.902,-179.651,8.349,149.505
C04419=1109.367,119.418,-59.919,-179.649,8.353,149.505
C04420=1109.363,119.632,-59.937,-179.647,8.355,149.505
C04421=1109.358,119.881,-59.958,-179.645,8.359,149.506
C04422=1109.353,120.130,-59.978,-179.644,8.362,149.506
C04423=1109.349,120.379,-59.998,-179.642,8.366,149.506
C04424=1109.344,120.629,-60.019,-179.640,8.369,149.507
C04425=1109.339,120.877,-60.040,-179.639,8.372,149.507
C04426=1109.335,121.126,-60.060,-179.637,8.376,149.507
C04427=1109.330,121.376,-60.081,-179.635,8.379,149.507
C04428=1109.325,121.625,-60.101,-179.634,8.382,149.508
C04429=1109.321,121.874,-60.122,-179.632,8.385,149.508
C04430=1109.316,122.123,-60.143,-179.630,8.389,149.508
C04431=1109.312,122.373,-60.164,-179.629,8.392,149.509
C04432=1109.307,122.622,-60.184,-179.627,8.395,149.509
C04433=1109.302,122.871,-60.205,-179.624,8.399,149.509
C04434=1109.298,123.120,-60.225,-179.623,8.402,149.510
C04435=1109.293,123.369,-60.246,-179.621,8.406,149.510
C04436=1109.288,123.618,-60.267,-179.619,8.409,149.510
C04437=1109.283,123.867,-60.288,-179.617,8.413,149.510
C04438=1109.279,124.116,-60.308,-179.616,8.416,149.511
C04439=1109.273,124.365,-60.329,-179.614,8.419,149.511
C04440=1109.269,124.614,-60.349,-179.612,8.423,149.511
C04441=1109.264,124.863,-60.371,-179.611,8.425,149.511
C04442=1109.260,125.112,-60.391,-179.609,8.429,149.512
C04443=1109.255,125.361,-60.412,-179.607,8.433,149.512
C04444=1109.251,125.611,-60.433,-179.606,8.435,149.512
C04445=1109.246,125.860,-60.454,-179.603,8.439,149.512
C04446=1109.241,126.109,-60.474,-179.602,8.443,149.513
C04447=1109.236,126.358,-60.495,-179.600,8.446,149.513
C04448=1109.232,126.607,-60.516,-179.598,8.449,149.513
C04449=1109.227,126.856,-60.537,-179.596,8.453,149.514
C04450=1109.222,127.105,-60.558,-179.595,8.455,149.514
C04451=1109.218,127.355,-60.579,-179.593,8.459,149.514
C04452=1109.213,127.604,-60.599,-179.591,8.463,149.514
C04453=1109.208,127.852,-60.621,-179.590,8.465,149.515
C04454=1109.204,128.101,-60.641,-179.588,8.469,149.515
C04455=1109.199,128.351,-60.662,-179.586,8.473,149.515
C04456=1109.194,128.599,-60.684,-179.585,8.475,149.516
C04457=1109.189,128.848,-60.705,-179.583,8.479,149.516
C04458=1109.185,129.098,-60.726,-179.580,8.482,149.516
C04459=1109.180,129.347,-60.747,-179.579,8.486,149.516
C04460=1109.176,129.596,-60.768,-179.577,8.489,149.517
C04461=1109.170,129.845,-60.789,-179.575,8.492,149.517
C04462=1109.166,130.094,-60.809,-179.573,8.496,149.517
C04463=1109.161,130.343,-60.831,-179.572,8.499,149.518
C04464=1109.156,130.593,-60.852,-179.570,8.503,149.518
C04465=1109.152,130.841,-60.873,-179.568,8.506,149.518
C04466=1109.147,131.090,-60.894,-179.567,8.509,149.518
C04467=1109.142,131.339,-60.915,-179.565,8.513,149.519
C04468=1109.138,131.588,-60.936,-179.563,8.516,149.519
C04469=1109.133,131.802,-60.955,-179.562,8.519,149.519
C04470=1109.130,132.016,-60.973,-179.560,8.522,149.519
C04471=1109.126,132.229,-60.991,-179.559,8.524,149.520
C04472=1109.122,132.442,-61.009,-179.557,8.527,149.520
C04473=1109.118,132.656,-61.028,-179.556,8.530,149.520
C04474=1109.113,132.870,-61.046,-179.554,8.534,149.521
C04475=1109.109,133.083,-61.064,-179.553,8.536,149.521
C04476=1109.105,133.296,-61.082,-179.551,8.539,149.521
C04477=1109.101,133.546,-61.104,-179.549,8.543,149.521
C04478=1109.096,133.795,-61.125,-179.548,8.545,149.521
C04479=1109.092,134.043,-61.146,-179.546,8.549,149.522
C04480=1109.087,134.292,-61.167,-179.544,8.553,149.522
C04481=1109.082,134.542,-61.189,-179.543,8.555,149.522
C04482=1109.077,134.791,-61.210,-179.541,8.559,149.523
C04483=1109.073,135.039,-61.231,-179.539,8.563,149.523
C04484=1109.069,135.289,-61.252,-179.537,8.565,149.523
C04485=1109.064,135.538,-61.274,-179.535,8.569,149.524
C04486=1109.058,135.787,-61.295,-179.534,8.573,149.524
C04487=1109.054,136.036,-61.317,-179.532,8.575,149.524
C04488=1109.050,136.285,-61.338,-179.530,8.579,149.524
C04489=1109.045,136.534,-61.359,-179.529,8.583,149.525
C04490=1109.040,136.783,-61.381,-179.527,8.586,149.525
C04491=1109.036,137.032,-61.403,-179.525,8.589,149.525
C04492=1109.031,137.281,-61.424,-179.523,8.593,149.526
C04493=1109.026,137.530,-61.445,-179.521,8.596,149.526
C04494=1109.022,137.779,-61.467,-179.520,8.599,149.526
C04495=1109.017,138.028,-61.488,-179.518,8.603,149.527
C04496=1109.012,138.277,-61.510,-179.516,8.606,149.527
C04497=1109.008,138.526,-61.532,-179.515,8.609,149.527
C04498=1109.003,138.775,-61.553,-179.513,8.613,149.528
C04499=1108.998,139.024,-61.574,-179.511,8.617,149.528
C04500=1108.994,139.274,-61.596,-179.509,8.620,149.528
C04501=1108.989,139.522,-61.618,-179.508,8.623,149.528
C04502=1108.984,139.772,-61.640,-179.506,8.627,149.529
C04503=1108.979,140.021,-61.661,-179.504,8.630,149.529
C04504=1108.975,140.269,-61.682,-179.503,8.633,149.529
C04505=1108.971,140.518,-61.704,-179.501,8.637,149.530
C04506=1108.966,140.767,-61.726,-179.499,8.641,149.530
C04507=1108.962,141.016,-61.748,-179.498,8.643,149.530
C04508=1108.957,141.266,-61.769,-179.496,8.647,149.531
C04509=1108.952,141.514,-61.791,-179.494,8.651,149.531
C04510=1108.947,141.764,-61.813,-179.492,8.654,149.531
C04511=1108.943,142.012,-61.834,-179.491,8.657,149.532
C04512=1108.938,142.262,-61.856,-179.489,8.661,149.532
C04513=1108.933,142.510,-61.878,-179.487,8.664,149.532
C04514=1108.929,142.760,-61.900,-179.485,8.668,149.533
C04515=1108.924,143.008,-61.922,-179.484,8.671,149.533
C04516=1108.919,143.257,-61.943,-179.482,8.675,149.533
C04517=1108.915,143.507,-61.965,-179.480,8.678,149.533
C04518=1108.910,143.756,-61.986,-179.479,8.681,149.534
C04519=1108.906,144.005,-62.008,-179.477,8.685,149.534
C04520=1108.901,144.254,-62.030,-179.475,8.688,149.534
C04521=1108.897,144.503,-62.052,-179.473,8.692,149.535
C04522=1108.892,144.751,-62.074,-179.472,8.695,149.535
C04523=1108.887,145.001,-62.097,-179.470,8.699,149.535
C04524=1108.882,145.250,-62.118,-179.468,8.702,149.536
C04525=1108.879,145.463,-62.137,-179.467,8.705,149.536
C04526=1108.874,145.677,-62.156,-179.465,8.709,149.536
C04527=1108.870,145.890,-62.174,-179.463,8.711,149.537
C04528=1108.866,146.103,-62.194,-179.461,8.715,149.537
C04529=1108.862,146.316,-62.212,-179.460,8.718,149.537
C04530=1108.858,146.531,-62.231,-179.458,8.720,149.537
C04531=1108.855,146.743,-62.250,-179.456,8.724,149.538
C04532=1108.851,146.957,-62.269,-179.455,8.727,149.538
C04533=1108.846,147.206,-62.291,-179.453,8.730,149.538
C04534=1108.841,147.455,-62.313,-179.451,8.734,149.538
C04535=1108.837,147.704,-62.335,-179.449,8.737,149.539
C04536=1108.832,147.953,-62.358,-179.447,8.741,149.539
C04537=1108.827,148.202,-62.380,-179.445,8.744,149.539
C04538=1108.823,148.451,-62.402,-179.443,8.748,149.539
C04539=1108.818,148.700,-62.423,-179.441,8.751,149.540
C04540=1108.814,148.949,-62.445,-179.439,8.755,149.540
C04541=1108.808,149.198,-62.468,-179.437,8.758,149.540
C04542=1108.804,149.447,-62.490,-179.435,8.762,149.541
C04543=1108.800,149.696,-62.513,-179.434,8.765,149.541
C04544=1108.795,149.945,-62.534,-179.431,8.768,149.541
C04545=1108.790,150.194,-62.557,-179.429,8.772,149.541
C04546=1108.785,150.442,-62.579,-179.427,8.775,149.542
C04547=1108.781,150.692,-62.601,-179.425,8.779,149.542
C04548=1108.776,150.940,-62.623,-179.423,8.782,149.542
C04549=1108.772,151.189,-62.646,-179.421,8.786,149.542
C04550=1108.767,151.439,-62.668,-179.419,8.789,149.542
C04551=1108.762,151.687,-62.690,-179.417,8.793,149.543
C04552=1108.757,151.937,-62.713,-179.415,8.796,149.543
C04553=1108.753,152.185,-62.735,-179.413,8.799,149.543
C04554=1108.749,152.434,-62.757,-179.411,8.802,149.543
C04555=1108.744,152.683,-62.781,-179.409,8.806,149.543
C04556=1108.739,152.932,-62.802,-179.407,8.809,149.544
C04557=1108.735,153.181,-62.824,-179.405,8.813,149.544
C04558=1108.730,153.430,-62.848,-179.403,8.816,149.544
C04559=1108.725,153.679,-62.869,-179.401,8.819,149.544
C04560=1108.721,153.928,-62.892,-179.399,8.822,149.545
C04561=1108.716,154.177,-62.915,-179.397,8.826,149.545
C04562=1108.711,154.426,-62.936,-179.394,8.829,149.545
C04563=1108.707,154.675,-62.959,-179.392,8.832,149.545
C04564=1108.702,154.924,-62.982,-179.390,8.836,149.545
C04565=1108.698,155.172,-63.004,-179.389,8.839,149.546
C04566=1108.693,155.422,-63.027,-179.387,8.842,149.546
C04567=1108.689,155.671,-63.050,-179.384,8.845,149.546
C04568=1108.684,155.919,-63.071,-179.382,8.849,149.546
C04569=1108.679,156.168,-63.095,-179.380,8.852,149.546
C04570=1108.675,156.417,-63.117,-179.378,8.856,149.547
C04571=1108.670,156.667,-63.140,-179.376,8.858,149.547
C04572=1108.666,156.915,-63.162,-179.374,8.861,149.547
C04573=1108.661,157.164,-63.185,-179.372,8.865,149.547
C04574=1108.657,157.413,-63.208,-179.369,8.868,149.547
C04575=1108.651,157.662,-63.230,-179.368,8.871,149.547
C04576=1108.647,157.911,-63.253,-179.366,8.874,149.548
C04577=1108.642,158.160,-63.276,-179.363,8.877,149.548
C04578=1108.638,158.409,-63.298,-179.361,8.881,149.548
C04579=1108.633,158.658,-63.321,-179.359,8.884,149.548
C04580=1108.629,158.906,-63.344,-179.357,8.887,149.548
C04581=1108.625,159.120,-63.364,-179.355,8.890,149.548
C04582=1108.621,159.333,-63.383,-179.353,8.892,149.548
C04583=1108.617,159.547,-63.402,-179.352,8.895,149.549
C04584=1108.613,159.760,-63.422,-179.350,8.898,149.549
C04585=1108.609,159.973,-63.442,-179.348,8.900,149.549
C04586=1108.606,160.186,-63.461,-179.346,8.904,149.549
C04587=1108.602,160.400,-63.481,-179.344,8.906,149.549
C04588=1108.597,160.613,-63.500,-179.343,8.909,149.549
C04589=1108.593,160.862,-63.523,-179.340,8.912,149.549
C04590=1108.589,161.111,-63.546,-179.338,8.915,149.550
C04591=1108.584,161.360,-63.569,-179.337,8.918,149.550
C04592=1108.578,161.609,-63.592,-179.334,8.921,149.550
C04593=1108.574,161.857,-63.615,-179.332,8.924,149.550
C04594=1108.570,162.106,-63.638,-179.330,8.928,149.550
C04595=1108.566,162.355,-63.661,-179.328,8.930,149.550
C04596=1108.561,162.604,-63.684,-179.326,8.934,149.551
C04597=1108.556,162.854,-63.707,-179.323,8.937,149.551
C04598=1108.552,163.103,-63.729,-179.322,8.939,149.551
C04599=1108.547,163.351,-63.752,-179.319,8.942,149.551
C04600=1108.542,163.600,-63.776,-179.317,8.946,149.551
C04601=1108.538,163.849,-63.799,-179.315,8.949,149.551
C04602=1108.533,164.098,-63.822,-179.313,8.952,149.551
C04603=1108.529,164.347,-63.845,-179.311,8.955,149.551
C04604=1108.525,164.595,-63.868,-179.309,8.958,149.552
C04605=1108.520,164.844,-63.891,-179.307,8.961,149.552
C04606=1108.515,165.093,-63.914,-179.305,8.964,149.552
C04607=1108.510,165.342,-63.938,-179.302,8.967,149.552
C04608=1108.506,165.590,-63.961,-179.300,8.971,149.552
C04609=1108.501,165.840,-63.984,-179.298,8.973,149.552
C04610=1108.497,166.089,-64.007,-179.296,8.976,149.552
C04611=1108.492,166.338,-64.031,-179.294,8.980,149.552
C04612=1108.488,166.586,-64.053,-179.292,8.982,149.553
C04613=1108.483,166.835,-64.077,-179.290,8.986,149.553
C04614=1108.479,167.084,-64.100,-179.287,8.989,149.553
C04615=1108.474,167.333,-64.123,-179.286,8.991,149.553
C04616=1108.470,167.582,-64.146,-179.283,8.994,149.553
C04617=1108.465,167.830,-64.169,-179.281,8.998,149.553
C04618=1108.460,168.079,-64.193,-179.279,9.000,149.553
C04619=1108.455,168.329,-64.216,-179.277,9.003,149.553
C04620=1108.451,168.578,-64.239,-179.275,9.007,149.554
C04621=1108.446,168.827,-64.263,-179.273,9.009,149.554
C04622=1108.442,169.075,-64.286,-179.270,9.012,149.554
C04623=1108.438,169.324,-64.310,-179.268,9.016,149.554
C04624=1108.433,169.573,-64.333,-179.266,9.018,149.554
C04625=1108.428,169.822,-64.356,-179.264,9.021,149.554
C04626=1108.423,170.071,-64.380,-179.262,9.025,149.554
C04627=1108.419,170.320,-64.403,-179.260,9.027,149.554
C04628=1108.414,170.568,-64.427,-179.257,9.030,149.554
C04629=1108.410,170.817,-64.450,-179.255,9.034,149.555
C04630=1108.406,171.066,-64.473,-179.253,9.036,149.555
C04631=1108.401,171.315,-64.496,-179.251,9.039,149.555
C04632=1108.397,171.563,-64.521,-179.249,9.043,149.555
C04633=1108.392,171.813,-64.544,-179.247,9.045,149.555
C04634=1108.387,172.062,-64.567,-179.245,9.048,149.555
C04635=1108.383,172.310,-64.591,-179.242,9.052,149.555
C04636=1108.378,172.559,-64.615,-179.240,9.054,149.555
C04637=1108.374,172.773,-64.635,-179.238,9.057,149.555
C04638=1108.370,172.986,-64.656,-179.236,9.060,149.556
C04639=1108.366,173.199,-64.675,-179.234,9.062,149.556
C04640=1108.362,173.412,-64.696,-179.232,9.064,149.556
C04641=1108.359,173.625,-64.715,-179.231,9.067,149.556
C04642=1108.355,173.838,-64.736,-179.229,9.069,149.556
C04643=1108.351,174.052,-64.756,-179.227,9.072,149.556
C04644=1108.347,174.265,-64.777,-179.225,9.075,149.556
C04645=1108.342,174.514,-64.800,-179.223,9.078,149.556
C04646=1108.338,174.762,-64.824,-179.221,9.081,149.556
C04647=1108.333,175.011,-64.848,-179.218,9.084,149.556
C04648=1108.329,175.260,-64.871,-179.217,9.086,149.556
C04649=1108.324,175.509,-64.895,-179.214,9.090,149.557
C04650=1108.319,175.758,-64.918,-179.212,9.092,149.557
C04651=1108.315,176.006,-64.942,-179.210,9.095,149.557
C04652=1108.311,176.256,-64.966,-179.208,9.098,149.557
C04653=1108.307,176.504,-64.990,-179.206,9.101,149.557
C04654=1108.302,176.753,-65.014,-179.204,9.104,149.557
C04655=1108.297,177.002,-65.038,-179.201,9.107,149.557
C04656=1108.292,177.251,-65.062,-179.199,9.110,149.557
C04657=1108.288,177.500,-65.086,-179.197,9.113,149.557
C04658=1108.283,177.748,-65.110,-179.195,9.116,149.557
C04659=1108.279,177.997,-65.133,-179.193,9.119,149.558
C04660=1108.275,178.246,-65.158,-179.191,9.122,149.558
C04661=1108.270,178.495,-65.181,-179.188,9.125,149.558
C04662=1108.266,178.744,-65.205,-179.186,9.128,149.558
C04663=1108.261,178.993,-65.228,-179.184,9.131,149.558
C04664=1108.257,179.241,-65.252,-179.182,9.134,149.558
C04665=1108.251,179.490,-65.277,-179.180,9.137,149.558
C04666=1108.247,179.739,-65.301,-179.177,9.140,149.558
C04667=1108.243,179.988,-65.325,-179.175,9.143,149.558
C04668=1108.239,180.236,-65.349,-179.173,9.146,149.559
C04669=1108.234,180.485,-65.372,-179.171,9.149,149.559
C04670=1108.229,180.734,-65.397,-179.168,9.152,149.559
C04671=1108.225,180.983,-65.421,-179.166,9.155,149.559
C04672=1108.221,181.232,-65.446,-179.163,9.158,149.559
C04673=1108.216,181.481,-65.469,-179.162,9.161,149.559
C04674=1108.211,181.729,-65.493,-179.159,9.164,149.559
C04675=1108.206,181.978,-65.518,-179.157,9.167,149.559
C04676=1108.203,182.227,-65.542,-179.154,9.170,149.559
C04677=1108.198,182.476,-65.565,-179.152,9.172,149.559
C04678=1108.193,182.724,-65.590,-179.150,9.175,149.559
C04679=1108.188,182.973,-65.614,-179.147,9.178,149.559
C04680=1108.185,183.222,-65.639,-179.145,9.182,149.559
C04681=1108.180,183.471,-65.663,-179.143,9.184,149.559
C04682=1108.175,183.720,-65.687,-179.140,9.187,149.559
C04683=1108.170,183.968,-65.711,-179.138,9.190,149.559
C04684=1108.166,184.217,-65.735,-179.136,9.192,149.559
C04685=1108.161,184.466,-65.760,-179.133,9.196,149.559
C04686=1108.157,184.715,-65.784,-179.131,9.199,149.560
C04687=1108.153,184.963,-65.808,-179.129,9.201,149.560
C04688=1108.148,185.212,-65.833,-179.126,9.204,149.560
C04689=1108.144,185.461,-65.857,-179.124,9.207,149.560
C04690=1108.139,185.709,-65.881,-179.122,9.210,149.560
C04691=1108.135,185.959,-65.906,-179.119,9.213,149.560
C04692=1108.130,186.208,-65.930,-179.117,9.216,149.560
C04693=1108.126,186.420,-65.951,-179.115,9.218,149.560
C04694=1108.123,186.633,-65.972,-179.113,9.220,149.560
C04695=1108.118,186.846,-65.993,-179.111,9.223,149.560
C04696=1108.115,187.059,-66.014,-179.109,9.225,149.560
C04697=1108.111,187.273,-66.035,-179.107,9.227,149.560
C04698=1108.107,187.486,-66.056,-179.106,9.230,149.560
C04699=1108.103,187.699,-66.076,-179.104,9.232,149.560
C04700=1108.099,187.912,-66.097,-179.102,9.234,149.560
C04701=1108.094,188.161,-66.122,-179.099,9.238,149.560
C04702=1108.090,188.410,-66.147,-179.097,9.241,149.560
C04703=1108.086,188.658,-66.171,-179.095,9.243,149.560
C04704=1108.081,188.908,-66.196,-179.092,9.246,149.560
C04705=1108.077,189.156,-66.220,-179.090,9.249,149.560
C04706=1108.072,189.404,-66.245,-179.088,9.252,149.560
C04707=1108.068,189.653,-66.270,-179.085,9.255,149.560
C04708=1108.063,189.902,-66.294,-179.083,9.257,149.560
C04709=1108.058,190.151,-66.318,-179.081,9.260,149.560
C04710=1108.054,190.400,-66.343,-179.078,9.263,149.561
C04711=1108.050,190.648,-66.367,-179.077,9.266,149.561
C04712=1108.045,190.898,-66.392,-179.074,9.269,149.561
C04713=1108.041,191.146,-66.417,-179.072,9.271,149.561
C04714=1108.036,191.394,-66.442,-179.070,9.274,149.561
C04715=1108.032,191.643,-66.466,-179.067,9.277,149.561
C04716=1108.027,191.892,-66.491,-179.065,9.280,149.561
C04717=1108.023,192.141,-66.516,-179.063,9.283,149.561
C04718=1108.018,192.389,-66.541,-179.061,9.285,149.561
C04719=1108.013,192.638,-66.566,-179.058,9.288,149.561
C04720=1108.009,192.887,-66.590,-179.056,9.291,149.561
C04721=1108.005,193.135,-66.615,-179.054,9.294,149.561
C04722=1108.001,193.384,-66.640,-179.052,9.297,149.561
C04723=1107.996,193.633,-66.664,-179.050,9.299,149.561
C04724=1107.991,193.882,-66.690,-179.047,9.302,149.561
C04725=1107.987,194.130,-66.714,-179.045,9.306,149.561
C04726=1107.982,194.380,-66.739,-179.043,9.308,149.561
C04727=1107.978,194.628,-66.765,-179.040,9.311,149.562
C04728=1107.973,194.876,-66.789,-179.038,9.313,149.562
C04729=1107.969,195.126,-66.814,-179.036,9.317,149.562
C04730=1107.965,195.374,-66.839,-179.034,9.320,149.562
C04731=1107.960,195.623,-66.864,-179.032,9.322,149.562
C04732=1107.955,195.871,-66.889,-179.029,9.325,149.562
C04733=1107.951,196.120,-66.914,-179.027,9.329,149.562
C04734=1107.946,196.369,-66.938,-179.025,9.331,149.562
C04735=1107.942,196.618,-66.964,-179.023,9.334,149.562
C04736=1107.937,196.866,-66.989,-179.020,9.337,149.562
C04737=1107.933,197.115,-67.014,-179.019,9.340,149.562
C04738=1107.928,197.364,-67.038,-179.016,9.343,149.562
C04739=1107.924,197.612,-67.064,-179.013,9.346,149.563
C04740=1107.920,197.862,-67.089,-179.011,9.349,149.563
C04741=1107.916,198.110,-67.114,-179.008,9.352,149.563
C04742=1107.911,198.359,-67.139,-179.006,9.355,149.563
C04743=1107.906,198.607,-67.164,-179.004,9.358,149.563
C04744=1107.902,198.856,-67.190,-179.001,9.361,149.563
C04745=1107.898,199.104,-67.214,-178.999,9.363,149.563
C04746=1107.893,199.353,-67.240,-178.996,9.367,149.563
C04747=1107.888,199.602,-67.265,-178.993,9.370,149.563
C04748=1107.884,199.851,-67.290,-178.992,9.372,149.563
C04749=1107.880,200.063,-67.312,-178.989,9.375,149.563
C04750=1107.876,200.277,-67.334,-178.987,9.377,149.563
C04751=1107.873,200.490,-67.355,-178.985,9.379,149.563
C04752=1107.869,200.702,-67.377,-178.982,9.382,149.563
C04753=1107.865,200.915,-67.398,-178.980,9.384,149.563
C04754=1107.862,201.129,-67.420,-178.978,9.386,149.562
C04755=1107.858,201.341,-67.442,-178.975,9.390,149.563
C04756=1107.854,201.555,-67.463,-178.973,9.392,149.563
C04757=1107.850,201.803,-67.489,-178.970,9.395,149.562
C04758=1107.845,202.052,-67.514,-178.968,9.398,149.562
C04759=1107.840,202.301,-67.539,-178.965,9.401,149.562
C04760=1107.836,202.550,-67.565,-178.962,9.403,149.562
C04761=1107.831,202.798,-67.590,-178.959,9.406,149.562
C04762=1107.827,203.047,-67.616,-178.956,9.409,149.562
C04763=1107.823,203.295,-67.641,-178.954,9.412,149.562
C04764=1107.818,203.544,-67.666,-178.951,9.415,149.562
C04765=1107.814,203.793,-67.692,-178.948,9.418,149.562
C04766=1107.809,204.041,-67.717,-178.946,9.420,149.562
C04767=1107.805,204.290,-67.743,-178.943,9.424,149.562
C04768=1107.801,204.538,-67.768,-178.940,9.426,149.562
C04769=1107.797,204.787,-67.794,-178.937,9.429,149.561
C04770=1107.792,205.035,-67.820,-178.934,9.432,149.562
C04771=1107.787,205.285,-67.845,-178.931,9.435,149.561
C04772=1107.783,205.534,-67.870,-178.928,9.438,149.561
C04773=1107.778,205.782,-67.896,-178.925,9.440,149.561
C04774=1107.774,206.031,-67.922,-178.923,9.443,149.561
C04775=1107.770,206.279,-67.947,-178.920,9.446,149.561
C04776=1107.764,206.528,-67.973,-178.917,9.449,149.561
C04777=1107.760,206.777,-67.999,-178.914,9.452,149.561
C04778=1107.756,207.025,-68.025,-178.911,9.454,149.561
C04779=1107.751,207.274,-68.051,-178.908,9.458,149.561
C04780=1107.747,207.522,-68.076,-178.905,9.461,149.561
C04781=1107.742,207.771,-68.102,-178.902,9.464,149.560
C04782=1107.738,208.020,-68.127,-178.899,9.467,149.560
C04783=1107.734,208.269,-68.153,-178.896,9.470,149.560
C04784=1107.729,208.517,-68.179,-178.893,9.473,149.560
C04785=1107.725,208.765,-68.205,-178.890,9.476,149.560
C04786=1107.720,209.014,-68.231,-178.887,9.479,149.560
C04787=1107.716,209.263,-68.257,-178.883,9.482,149.560
C04788=1107.711,209.511,-68.282,-178.881,9.485,149.560
C04789=1107.707,209.760,-68.308,-178.878,9.488,149.560
C04790=1107.703,210.009,-68.334,-178.874,9.492,149.560
C04791=1107.699,210.257,-68.360,-178.872,9.495,149.560
C04792=1107.694,210.506,-68.387,-178.869,9.497,149.560
C04793=1107.690,210.755,-68.413,-178.865,9.501,149.559
C04794=1107.685,211.003,-68.438,-178.862,9.504,149.559
C04795=1107.681,211.252,-68.464,-178.859,9.508,149.559
C04796=1107.677,211.500,-68.490,-178.856,9.510,149.559
C04797=1107.672,211.749,-68.517,-178.853,9.514,149.559
C04798=1107.667,211.998,-68.542,-178.850,9.517,149.559
C04799=1107.663,212.247,-68.568,-178.847,9.521,149.559
C04800=1107.659,212.494,-68.594,-178.844,9.524,149.559
C04801=1107.654,212.743,-68.620,-178.840,9.527,149.559
C04802=1107.650,212.991,-68.647,-178.838,9.530,149.559
C04803=1107.646,213.240,-68.673,-178.834,9.534,149.559
C04804=1107.641,213.489,-68.699,-178.831,9.537,149.559
C04805=1107.638,213.702,-68.722,-178.829,9.540,149.559
C04806=1107.634,213.915,-68.744,-178.827,9.542,149.559
C04807=1107.629,214.127,-68.766,-178.826,9.545,149.559
C04808=1107.626,214.340,-68.789,-178.824,9.547,149.559
C04809=1107.622,214.553,-68.811,-178.821,9.550,149.559
C04810=1107.618,214.766,-68.834,-178.819,9.552,149.559
C04811=1107.615,214.978,-68.856,-178.817,9.555,149.559
C04812=1107.611,215.192,-68.878,-178.816,9.558,149.560
C04813=1107.607,215.440,-68.906,-178.813,9.561,149.560
C04814=1107.602,215.689,-68.931,-178.811,9.564,149.560
C04815=1107.598,215.938,-68.958,-178.808,9.567,149.560
C04816=1107.594,216.186,-68.984,-178.806,9.569,149.560
C04817=1107.590,216.435,-69.011,-178.804,9.573,149.560
C04818=1107.585,216.684,-69.037,-178.802,9.576,149.560
C04819=1107.581,216.932,-69.063,-178.799,9.579,149.560
C04820=1107.576,217.181,-69.090,-178.797,9.581,149.560
C04821=1107.572,217.429,-69.116,-178.795,9.584,149.560
C04822=1107.568,217.677,-69.143,-178.793,9.588,149.561
C04823=1107.563,217.926,-69.169,-178.790,9.591,149.561
C04824=1107.559,218.175,-69.195,-178.788,9.594,149.561
C04825=1107.554,218.424,-69.222,-178.786,9.596,149.561
C04826=1107.550,218.672,-69.248,-178.784,9.600,149.561
C04827=1107.546,218.920,-69.275,-178.781,9.603,149.561
C04828=1107.541,219.169,-69.301,-178.779,9.606,149.561
C04829=1107.537,219.418,-69.328,-178.776,9.609,149.561
C04830=1107.533,219.666,-69.355,-178.774,9.612,149.561
C04831=1107.528,219.915,-69.381,-178.772,9.615,149.562
C04832=1107.524,220.163,-69.407,-178.770,9.618,149.562
C04833=1107.519,220.412,-69.434,-178.767,9.621,149.562
C04834=1107.515,220.660,-69.461,-178.765,9.624,149.562
C04835=1107.510,220.909,-69.487,-178.762,9.627,149.562
C04836=1107.506,221.158,-69.514,-178.759,9.631,149.562
C04837=1107.502,221.406,-69.541,-178.758,9.633,149.562
C04838=1107.497,221.654,-69.568,-178.755,9.636,149.562
C04839=1107.493,221.902,-69.594,-178.753,9.639,149.562
C04840=1107.488,222.152,-69.621,-178.750,9.643,149.562
C04841=1107.484,222.400,-69.647,-178.748,9.646,149.562
C04842=1107.480,222.648,-69.674,-178.745,9.649,149.563
C04843=1107.475,222.897,-69.701,-178.743,9.652,149.563
C04844=1107.471,223.145,-69.728,-178.741,9.655,149.563
C04845=1107.467,223.394,-69.755,-178.739,9.658,149.563
C04846=1107.462,223.643,-69.782,-178.736,9.661,149.563
C04847=1107.458,223.891,-69.808,-178.734,9.664,149.563
C04848=1107.453,224.140,-69.835,-178.731,9.667,149.563
C04849=1107.449,224.388,-69.862,-178.729,9.670,149.563
C04850=1107.445,224.637,-69.889,-178.727,9.672,149.563
C04851=1107.440,224.885,-69.916,-178.724,9.676,149.563
C04852=1107.436,225.134,-69.943,-178.722,9.679,149.563
C04853=1107.432,225.382,-69.969,-178.719,9.682,149.563
C04854=1107.428,225.631,-69.997,-178.717,9.685,149.564
C04855=1107.423,225.879,-70.024,-178.714,9.688,149.564
C04856=1107.419,226.128,-70.050,-178.712,9.691,149.564
C04857=1107.414,226.376,-70.077,-178.710,9.693,149.564
C04858=1107.410,226.625,-70.104,-178.707,9.696,149.564
C04859=1107.405,226.873,-70.131,-178.704,9.699,149.564
C04860=1107.402,227.122,-70.158,-178.702,9.702,149.564
C04861=1107.397,227.334,-70.181,-178.700,9.705,149.564
C04862=1107.394,227.547,-70.205,-178.697,9.708,149.564
C04863=1107.390,227.760,-70.228,-178.696,9.710,149.564
C04864=1107.386,227.972,-70.251,-178.694,9.713,149.564
C04865=1107.383,228.185,-70.274,-178.691,9.715,149.564
C04866=1107.379,228.398,-70.298,-178.689,9.718,149.564
C04867=1107.375,228.610,-70.320,-178.687,9.720,149.564
C04868=1107.372,228.823,-70.344,-178.685,9.722,149.564
C04869=1107.367,229.072,-70.371,-178.682,9.725,149.564
C04870=1107.363,229.321,-70.398,-178.680,9.728,149.564
C04871=1107.358,229.569,-70.426,-178.677,9.731,149.564
C04872=1107.354,229.817,-70.453,-178.675,9.733,149.564
C04873=1107.350,230.066,-70.480,-178.672,9.736,149.564
C04874=1107.345,230.314,-70.507,-178.669,9.739,149.564
C04875=1107.342,230.563,-70.535,-178.667,9.742,149.564
C04876=1107.337,230.811,-70.562,-178.664,9.745,149.564
C04877=1107.332,231.060,-70.589,-178.662,9.747,149.564
C04878=1107.328,231.308,-70.616,-178.659,9.750,149.564
C04879=1107.324,231.557,-70.644,-178.656,9.753,149.564
C04880=1107.319,231.805,-70.671,-178.653,9.756,149.564
C04881=1107.314,232.054,-70.698,-178.652,9.758,149.564
C04882=1107.311,232.302,-70.726,-178.649,9.761,149.564
C04883=1107.307,232.551,-70.753,-178.646,9.764,149.563
C04884=1107.302,232.799,-70.780,-178.643,9.767,149.564
C04885=1107.298,233.047,-70.808,-178.641,9.769,149.563
C04886=1107.294,233.296,-70.835,-178.638,9.772,149.563
C04887=1107.289,233.545,-70.862,-178.635,9.775,149.563
C04888=1107.285,233.792,-70.890,-178.633,9.777,149.563
C04889=1107.281,234.042,-70.917,-178.630,9.779,149.563
C04890=1107.276,234.290,-70.945,-178.628,9.783,149.563
C04891=1107.272,234.538,-70.972,-178.625,9.785,149.563
C04892=1107.268,234.787,-71.000,-178.622,9.787,149.563
C04893=1107.263,235.035,-71.028,-178.620,9.790,149.563
C04894=1107.259,235.283,-71.055,-178.617,9.793,149.563
C04895=1107.255,235.532,-71.083,-178.615,9.795,149.563
C04896=1107.251,235.780,-71.110,-178.612,9.798,149.563
C04897=1107.246,236.029,-71.138,-178.609,9.801,149.563
C04898=1107.242,236.277,-71.166,-178.607,9.803,149.563
C04899=1107.237,236.526,-71.193,-178.604,9.806,149.562
C04900=1107.232,236.774,-71.221,-178.601,9.808,149.562
C04901=1107.228,237.023,-71.249,-178.599,9.810,149.562
C04902=1107.224,237.271,-71.276,-178.596,9.814,149.562
C04903=1107.220,237.519,-71.304,-178.593,9.816,149.562
C04904=1107.216,237.768,-71.332,-178.590,9.819,149.562
C04905=1107.211,238.016,-71.359,-178.588,9.821,149.562
C04906=1107.207,238.265,-71.387,-178.585,9.824,149.562
C04907=1107.203,238.513,-71.415,-178.582,9.827,149.562
C04908=1107.198,238.762,-71.443,-178.580,9.829,149.562
C04909=1107.194,239.010,-71.470,-178.577,9.832,149.562
C04910=1107.189,239.258,-71.498,-178.574,9.834,149.561
C04911=1107.186,239.507,-71.526,-178.572,9.837,149.561
C04912=1107.181,239.755,-71.554,-178.569,9.839,149.561
C04913=1107.177,240.004,-71.581,-178.566,9.842,149.561
C04914=1107.172,240.252,-71.610,-178.564,9.844,149.561
C04915=1107.168,240.501,-71.638,-178.562,9.847,149.561
C04916=1107.164,240.748,-71.666,-178.559,9.850,149.561
C04917=1107.160,240.961,-71.689,-178.556,9.852,149.561
C04918=1107.157,241.174,-71.713,-178.554,9.854,149.561
C04919=1107.153,241.387,-71.737,-178.552,9.856,149.561
C04920=1107.150,241.599,-71.761,-178.550,9.858,149.561
C04921=1107.146,241.812,-71.785,-178.547,9.861,149.561
C04922=1107.142,242.024,-71.809,-178.545,9.863,149.561
C04923=1107.138,242.237,-71.833,-178.543,9.866,149.561
C04924=1107.134,242.450,-71.857,-178.541,9.868,149.561
C04925=1107.130,242.698,-71.885,-178.538,9.870,149.560
C04926=1107.126,242.946,-71.913,-178.535,9.874,149.561
C04927=1107.122,243.195,-71.941,-178.533,9.875,149.560
C04928=1107.117,243.443,-71.969,-178.530,9.879,149.560
C04929=1107.113,243.691,-71.997,-178.527,9.881,149.560
C04930=1107.109,243.939,-72.025,-178.525,9.884,149.560
C04931=1107.104,244.188,-72.054,-178.523,9.886,149.560
C04932=1107.100,244.436,-72.082,-178.520,9.889,149.560
C04933=1107.096,244.685,-72.110,-178.517,9.892,149.560
C04934=1107.091,244.933,-72.138,-178.514,9.895,149.560
C04935=1107.087,245.182,-72.166,-178.512,9.897,149.560
C04936=1107.083,245.430,-72.193,-178.509,9.900,149.560
C04937=1107.079,245.678,-72.223,-178.507,9.903,149.560
C04938=1107.075,245.927,-72.251,-178.504,9.906,149.560
C04939=1107.070,246.175,-72.279,-178.501,9.909,149.560
C04940=1107.066,246.424,-72.308,-178.499,9.911,149.560
C04941=1107.062,246.671,-72.335,-178.497,9.914,149.560
C04942=1107.057,246.920,-72.364,-178.494,9.917,149.560
C04943=1107.053,247.168,-72.392,-178.491,9.920,149.560
C04944=1107.048,247.417,-72.421,-178.489,9.924,149.560
C04945=1107.045,247.666,-72.449,-178.486,9.926,149.560
C04946=1107.040,247.914,-72.477,-178.483,9.929,149.560
C04947=1107.036,248.162,-72.505,-178.481,9.931,149.560
C04948=1107.032,248.410,-72.534,-178.479,9.935,149.560
C04949=1107.027,248.659,-72.562,-178.476,9.937,149.560
C04950=1107.024,248.907,-72.591,-178.473,9.940,149.560
C04951=1107.018,249.155,-72.619,-178.470,9.943,149.560
C04952=1107.015,249.404,-72.647,-178.467,9.946,149.560
C04953=1107.011,249.652,-72.677,-178.465,9.948,149.560
C04954=1107.006,249.900,-72.704,-178.462,9.951,149.560
C04955=1107.002,250.149,-72.733,-178.459,9.953,149.560
C04956=1106.998,250.398,-72.761,-178.456,9.956,149.560
C04957=1106.993,250.645,-72.790,-178.454,9.958,149.559
C04958=1106.989,250.894,-72.819,-178.451,9.961,149.559
C04959=1106.985,251.143,-72.847,-178.448,9.964,149.559
C04960=1106.980,251.390,-72.876,-178.445,9.965,149.559
C04961=1106.976,251.639,-72.904,-178.442,9.968,149.559
C04962=1106.972,251.888,-72.933,-178.439,9.971,149.559
C04963=1106.968,252.135,-72.962,-178.437,9.973,149.558
C04964=1106.963,252.384,-72.990,-178.434,9.975,149.558
C04965=1106.959,252.633,-73.019,-178.431,9.978,149.558
C04966=1106.955,252.880,-73.048,-178.428,9.980,149.558
C04967=1106.950,253.129,-73.076,-178.426,9.983,149.558
C04968=1106.947,253.377,-73.105,-178.423,9.985,149.558
C04969=1106.942,253.625,-73.134,-178.420,9.987,149.557
C04970=1106.937,253.874,-73.162,-178.417,9.990,149.557
C04971=1106.934,254.122,-73.191,-178.414,9.992,149.557
C04972=1106.929,254.371,-73.220,-178.411,9.995,149.557
C04973=1106.926,254.592,-73.246,-178.409,9.997,149.557
C04974=1106.922,254.814,-73.271,-178.406,9.999,149.557
C04975=1106.917,255.036,-73.297,-178.403,10.002,149.557
C04976=1106.914,255.258,-73.323,-178.402,10.004,149.557
C04977=1106.910,255.480,-73.348,-178.399,10.006,149.557
C04978=1106.906,255.702,-73.374,-178.396,10.009,149.557
C04979=1106.902,255.924,-73.401,-178.394,10.011,149.556
C04980=1106.899,256.146,-73.426,-178.392,10.013,149.556
C04981=1106.895,256.394,-73.456,-178.389,10.016,149.556
C04982=1106.890,256.642,-73.484,-178.386,10.019,149.556
C04983=1106.886,256.891,-73.513,-178.384,10.022,149.556
C04984=1106.882,257.139,-73.542,-178.381,10.025,149.556
C04985=1106.642,246.650,-72.391,-178.495,9.915,149.560
C04986=1106.646,246.402,-72.363,-178.498,9.913,149.560
C04987=1106.651,246.154,-72.335,-178.500,9.910,149.560
C04988=1106.655,245.905,-72.305,-178.503,9.906,149.560
C04989=1106.659,245.657,-72.277,-178.506,9.904,149.560
C04990=1106.663,245.409,-72.249,-178.508,9.901,149.560
C04991=1106.667,245.160,-72.221,-178.511,9.899,149.560
C04992=1106.672,244.912,-72.193,-178.513,9.895,149.560
C04993=1106.676,244.663,-72.164,-178.516,9.893,149.560
C04994=1106.681,244.415,-72.136,-178.519,9.890,149.560
C04995=1106.684,244.167,-72.108,-178.521,9.888,149.560
C04996=1106.690,243.918,-72.081,-178.523,9.885,149.560
C04997=1106.694,243.669,-72.052,-178.526,9.882,149.560
C04998=1106.698,243.422,-72.025,-178.529,9.879,149.560
C04999=1106.702,243.173,-71.996,-178.531,9.877,149.560
C05000=1106.707,242.925,-71.968,-178.534,9.874,149.560
C05001=1106.710,242.676,-71.940,-178.537,9.871,149.560
C05002=1106.714,242.435,-71.913,-178.540,9.868,149.560
C05003=1106.719,242.195,-71.886,-178.542,9.866,149.561
C05004=1106.724,241.954,-71.859,-178.544,9.863,149.560
C05005=1106.727,241.714,-71.831,-178.547,9.861,149.561
C05006=1106.732,241.474,-71.804,-178.550,9.858,149.561
C05007=1106.736,241.233,-71.777,-178.552,9.855,149.561
C05008=1106.739,240.992,-71.750,-178.555,9.853,149.561
C05009=1106.744,240.752,-71.724,-178.558,9.850,149.561
C05010=1106.748,240.503,-71.695,-178.560,9.848,149.561
C05011=1106.753,240.255,-71.667,-178.562,9.845,149.561
C05012=1106.757,240.006,-71.640,-178.565,9.843,149.561
C05013=1106.761,239.758,-71.612,-178.568,9.840,149.561
C05014=1106.765,239.509,-71.584,-178.571,9.838,149.561
C05015=1106.770,239.261,-71.557,-178.573,9.835,149.561
C05016=1106.774,239.012,-71.528,-178.576,9.832,149.561
C05017=1106.778,238.764,-71.500,-178.578,9.830,149.561
C05018=1106.783,238.516,-71.472,-178.581,9.827,149.562
C05019=1106.787,238.267,-71.445,-178.584,9.825,149.562
C05020=1106.791,238.019,-71.417,-178.586,9.822,149.562
C05021=1106.795,237.770,-71.390,-178.589,9.819,149.562
C05022=1106.800,237.522,-71.362,-178.592,9.817,149.562
C05023=1106.805,237.274,-71.334,-178.594,9.815,149.562
C05024=1106.809,237.025,-71.306,-178.597,9.812,149.562
C05025=1106.813,236.777,-71.278,-178.600,9.809,149.562
C05026=1106.818,236.528,-71.251,-178.602,9.807,149.562
C05027=1106.821,236.280,-71.223,-178.605,9.804,149.562
C05028=1106.826,236.032,-71.195,-178.608,9.801,149.562
C05029=1106.830,235.783,-71.168,-178.611,9.798,149.562
C05030=1106.834,235.535,-71.140,-178.613,9.796,149.563
C05031=1106.839,235.286,-71.113,-178.616,9.794,149.563
C05032=1106.843,235.038,-71.085,-178.619,9.791,149.563
C05033=1106.847,234.789,-71.058,-178.621,9.788,149.563
C05034=1106.852,234.541,-71.030,-178.624,9.786,149.563
C05035=1106.856,234.292,-71.003,-178.626,9.783,149.563
C05036=1106.860,234.044,-70.976,-178.628,9.781,149.563
C05037=1106.865,233.796,-70.948,-178.631,9.778,149.563
C05038=1106.869,233.547,-70.920,-178.634,9.775,149.563
C05039=1106.873,233.299,-70.893,-178.636,9.773,149.563
C05040=1106.878,233.050,-70.866,-178.639,9.770,149.563
C05041=1106.882,232.802,-70.839,-178.642,9.767,149.563
C05042=1106.886,232.553,-70.810,-178.645,9.764,149.563
C05043=1106.891,232.305,-70.783,-178.647,9.762,149.563
C05044=1106.895,232.057,-70.756,-178.649,9.759,149.563
C05045=1106.899,231.808,-70.728,-178.652,9.756,149.563
C05046=1106.904,231.559,-70.701,-178.655,9.754,149.564
C05047=1106.908,231.311,-70.673,-178.657,9.751,149.564
C05048=1106.912,231.063,-70.647,-178.660,9.748,149.564
C05049=1106.916,230.814,-70.619,-178.663,9.745,149.564
C05050=1106.921,230.565,-70.592,-178.665,9.743,149.564
C05051=1106.925,230.318,-70.565,-178.668,9.740,149.564
C05052=1106.930,230.069,-70.538,-178.670,9.738,149.564
C05053=1106.934,229.820,-70.510,-178.673,9.734,149.564
C05054=1106.939,229.571,-70.483,-178.676,9.731,149.564
C05055=1106.943,229.323,-70.456,-178.678,9.729,149.564
C05056=1106.947,229.075,-70.429,-178.680,9.726,149.564
C05057=1106.951,228.826,-70.401,-178.683,9.723,149.564
C05058=1106.955,228.614,-70.378,-178.685,9.721,149.564
C05059=1106.959,228.401,-70.355,-178.687,9.719,149.564
C05060=1106.962,228.188,-70.332,-178.690,9.716,149.564
C05061=1106.966,227.976,-70.309,-178.692,9.713,149.564
C05062=1106.970,227.763,-70.285,-178.693,9.711,149.564
C05063=1106.974,227.550,-70.262,-178.696,9.709,149.564
C05064=1106.977,227.338,-70.239,-178.698,9.706,149.564
C05065=1106.981,227.125,-70.216,-178.700,9.704,149.564
C05066=1106.986,226.876,-70.189,-178.703,9.701,149.563
C05067=1106.990,226.628,-70.162,-178.705,9.697,149.563
C05068=1106.994,226.380,-70.135,-178.707,9.695,149.563
C05069=1106.998,226.130,-70.108,-178.710,9.692,149.563
C05070=1107.003,225.882,-70.081,-178.712,9.689,149.563
C05071=1107.007,225.634,-70.054,-178.715,9.686,149.563
C05072=1107.012,225.385,-70.027,-178.717,9.683,149.563
C05073=1107.016,225.137,-70.000,-178.720,9.680,149.563
C05074=1107.021,224.888,-69.973,-178.722,9.677,149.563
C05075=1107.024,224.639,-69.946,-178.724,9.674,149.563
C05076=1107.029,224.391,-69.919,-178.727,9.671,149.563
C05077=1107.034,224.142,-69.892,-178.729,9.668,149.563
C05078=1107.037,223.894,-69.865,-178.732,9.665,149.563
C05079=1107.042,223.646,-69.838,-178.734,9.662,149.563
C05080=1107.047,223.397,-69.811,-178.736,9.659,149.563
C05081=1107.051,223.148,-69.786,-178.739,9.656,149.562
C05082=1107.056,222.900,-69.759,-178.741,9.653,149.562
C05083=1107.060,222.652,-69.732,-178.744,9.650,149.562
C05084=1107.064,222.403,-69.705,-178.746,9.647,149.562
C05085=1107.068,222.154,-69.678,-178.749,9.644,149.562
C05086=1107.072,221.906,-69.651,-178.751,9.640,149.562
C05087=1107.077,221.657,-69.624,-178.753,9.638,149.562
C05088=1107.081,221.408,-69.598,-178.755,9.635,149.562
C05089=1107.086,221.160,-69.571,-178.758,9.632,149.562
C05090=1107.090,220.911,-69.544,-178.760,9.629,149.562
C05091=1107.094,220.663,-69.518,-178.763,9.625,149.562
C05092=1107.099,220.414,-69.491,-178.765,9.622,149.561
C05093=1107.103,220.166,-69.465,-178.767,9.620,149.561
C05094=1107.108,219.917,-69.438,-178.769,9.617,149.561
C05095=1107.112,219.669,-69.411,-178.772,9.613,149.561
C05096=1107.117,219.420,-69.385,-178.774,9.610,149.561
C05097=1107.121,219.172,-69.359,-178.777,9.607,149.561
C05098=1107.125,218.923,-69.331,-178.779,9.604,149.561
C05099=1107.130,218.675,-69.306,-178.781,9.601,149.561
C05100=1107.134,218.426,-69.279,-178.783,9.598,149.561
C05101=1107.138,218.178,-69.252,-178.786,9.595,149.561
C05102=1107.143,217.929,-69.226,-178.788,9.592,149.560
C05103=1107.147,217.681,-69.199,-178.791,9.589,149.560
C05104=1107.152,217.432,-69.172,-178.793,9.586,149.560
C05105=1107.156,217.183,-69.147,-178.795,9.583,149.560
C05106=1107.160,216.935,-69.120,-178.797,9.580,149.560
C05107=1107.165,216.686,-69.094,-178.800,9.577,149.560
C05108=1107.169,216.438,-69.067,-178.802,9.573,149.560
C05109=1107.174,216.189,-69.041,-178.804,9.571,149.560
C05110=1107.178,215.941,-69.014,-178.807,9.568,149.560
C05111=1107.182,215.692,-68.989,-178.809,9.565,149.559
C05112=1107.186,215.443,-68.962,-178.811,9.561,149.559
C05113=1107.191,215.195,-68.936,-178.813,9.559,149.559
C05114=1107.195,214.982,-68.913,-178.816,9.556,149.559
C05115=1107.198,214.769,-68.891,-178.818,9.554,149.559
C05116=1107.202,214.557,-68.868,-178.819,9.551,149.559
C05117=1107.206,214.343,-68.845,-178.821,9.549,149.559
C05118=1107.210,214.131,-68.823,-178.823,9.546,149.559
C05119=1107.213,213.918,-68.801,-178.825,9.543,149.559
C05120=1107.217,213.705,-68.778,-178.827,9.541,149.559
C05121=1107.221,213.492,-68.756,-178.829,9.539,149.559
C05122=1107.225,213.244,-68.730,-178.832,9.535,149.559
C05123=1107.230,212.995,-68.703,-178.835,9.532,149.559
C05124=1107.234,212.747,-68.677,-178.839,9.528,149.559
C05125=1107.238,212.498,-68.651,-178.842,9.524,149.559
C05126=1107.243,212.249,-68.625,-178.845,9.522,149.559
C05127=1107.247,212.001,-68.598,-178.848,9.518,149.559
C05128=1107.252,211.752,-68.573,-178.851,9.515,149.559
C05129=1107.256,211.503,-68.547,-178.855,9.512,149.559
C05130=1107.261,211.255,-68.522,-178.857,9.508,149.559
C05131=1107.265,211.007,-68.494,-178.861,9.505,149.559
C05132=1107.269,210.758,-68.469,-178.864,9.502,149.559
C05133=1107.274,210.509,-68.443,-178.867,9.499,149.559
C05134=1107.278,210.260,-68.417,-178.870,9.496,149.559
C05135=1107.283,210.012,-68.390,-178.873,9.492,149.559
C05136=1107.287,209.764,-68.365,-178.876,9.489,149.560
C05137=1107.292,209.515,-68.339,-178.879,9.487,149.560
C05138=1107.296,209.266,-68.313,-178.882,9.483,149.560
C05139=1107.300,209.017,-68.288,-178.885,9.480,149.560
C05140=1107.304,208.768,-68.262,-178.888,9.477,149.560
C05141=1107.309,208.520,-68.236,-178.892,9.474,149.560
C05142=1107.314,208.271,-68.210,-178.894,9.471,149.560
C05143=1107.318,208.023,-68.184,-178.897,9.468,149.560
C05144=1107.322,207.774,-68.158,-178.900,9.465,149.560
C05145=1107.327,207.526,-68.132,-178.903,9.462,149.560
C05146=1107.331,207.277,-68.107,-178.907,9.459,149.560
C05147=1107.335,207.028,-68.081,-178.909,9.456,149.560
C05148=1107.340,206.780,-68.055,-178.912,9.453,149.561
C05149=1107.345,206.531,-68.030,-178.915,9.450,149.561
C05150=1107.349,206.283,-68.004,-178.918,9.447,149.561
C05151=1107.353,206.034,-67.978,-178.921,9.444,149.561
C05152=1107.358,205.786,-67.953,-178.924,9.441,149.561
C05153=1107.362,205.537,-67.927,-178.927,9.438,149.561
C05154=1107.367,205.288,-67.902,-178.930,9.435,149.561
C05155=1107.371,205.039,-67.876,-178.933,9.432,149.561
C05156=1107.376,204.791,-67.851,-178.936,9.429,149.561
C05157=1107.380,204.542,-67.825,-178.939,9.427,149.561
C05158=1107.384,204.293,-67.800,-178.941,9.424,149.562
C05159=1107.389,204.045,-67.774,-178.944,9.421,149.562
C05160=1107.393,203.796,-67.748,-178.947,9.418,149.562
C05161=1107.397,203.547,-67.723,-178.950,9.415,149.562
C05162=1107.402,203.299,-67.698,-178.952,9.412,149.562
C05163=1107.407,203.050,-67.672,-178.955,9.410,149.562
C05164=1107.412,202.802,-67.647,-178.958,9.407,149.562
C05165=1107.416,202.553,-67.621,-178.961,9.404,149.562
C05166=1107.420,202.303,-67.596,-178.963,9.402,149.562
C05167=1107.425,202.055,-67.571,-178.966,9.399,149.562
C05168=1107.429,201.807,-67.545,-178.969,9.396,149.562
C05169=1107.434,201.558,-67.519,-178.971,9.393,149.562
C05170=1107.438,201.344,-67.498,-178.973,9.391,149.562
C05171=1107.442,201.132,-67.476,-178.976,9.388,149.562
C05172=1107.445,200.920,-67.455,-178.978,9.386,149.562
C05173=1107.448,200.706,-67.433,-178.980,9.383,149.562
C05174=1107.452,200.493,-67.412,-178.983,9.380,149.562
C05175=1107.456,200.280,-67.390,-178.985,9.378,149.562
C05176=1107.460,200.068,-67.368,-178.987,9.376,149.562
C05177=1107.464,199.854,-67.347,-178.989,9.373,149.562
C05178=1107.469,199.606,-67.321,-178.992,9.371,149.563
C05179=1107.473,199.356,-67.296,-178.994,9.368,149.563
C05180=1107.477,199.108,-67.271,-178.997,9.365,149.562
C05181=1107.481,198.860,-67.246,-178.999,9.362,149.562
C05182=1107.487,198.611,-67.221,-179.002,9.358,149.562
C05183=1107.491,198.362,-67.195,-179.004,9.356,149.562
C05184=1107.495,198.113,-67.170,-179.007,9.353,149.562
C05185=1107.499,197.865,-67.145,-179.009,9.350,149.562
C05186=1107.504,197.615,-67.120,-179.012,9.347,149.562
C05187=1107.509,197.367,-67.095,-179.014,9.344,149.562
C05188=1107.513,197.118,-67.070,-179.016,9.342,149.562
C05189=1107.517,196.870,-67.045,-179.019,9.339,149.562
C05190=1107.522,196.621,-67.020,-179.021,9.335,149.562
C05191=1107.527,196.373,-66.995,-179.023,9.332,149.562
C05192=1107.531,196.124,-66.970,-179.025,9.330,149.562
C05193=1107.535,195.875,-66.945,-179.028,9.327,149.562
C05194=1107.540,195.626,-66.920,-179.030,9.324,149.562
C05195=1107.544,195.378,-66.896,-179.032,9.321,149.561
C05196=1107.548,195.129,-66.870,-179.034,9.318,149.561
C05197=1107.554,194.880,-66.845,-179.036,9.315,149.561
C05198=1107.557,194.632,-66.820,-179.039,9.312,149.561
C05199=1107.562,194.383,-66.795,-179.041,9.309,149.561
C05200=1107.567,194.133,-66.770,-179.043,9.307,149.561
C05201=1107.571,193.886,-66.746,-179.045,9.303,149.561
C05202=1107.575,193.636,-66.721,-179.047,9.301,149.561
C05203=1107.581,193.387,-66.696,-179.050,9.298,149.561
C05204=1107.585,193.140,-66.671,-179.052,9.295,149.561
C05205=1107.589,192.890,-66.646,-179.054,9.292,149.561
C05206=1107.594,192.642,-66.622,-179.057,9.289,149.561
C05207=1107.598,192.393,-66.596,-179.058,9.287,149.561
C05208=1107.603,192.144,-66.572,-179.061,9.284,149.561
C05209=1107.607,191.895,-66.547,-179.064,9.281,149.561
C05210=1107.612,191.646,-66.523,-179.065,9.278,149.561
C05211=1107.616,191.399,-66.498,-179.068,9.275,149.561
C05212=1107.620,191.149,-66.473,-179.070,9.273,149.560
C05213=1107.625,190.901,-66.449,-179.072,9.270,149.560
C05214=1107.629,190.651,-66.424,-179.075,9.267,149.560
C05215=1107.634,190.403,-66.400,-179.077,9.264,149.560
C05216=1107.639,190.154,-66.375,-179.079,9.261,149.560
C05217=1107.642,189.906,-66.350,-179.082,9.258,149.560
C05218=1107.647,189.657,-66.325,-179.084,9.256,149.560
C05219=1107.651,189.408,-66.301,-179.086,9.253,149.560
C05220=1107.656,189.159,-66.276,-179.088,9.250,149.560
C05221=1107.661,188.911,-66.252,-179.091,9.247,149.560
C05222=1107.665,188.661,-66.227,-179.093,9.244,149.560
C05223=1107.670,188.413,-66.203,-179.095,9.242,149.560
C05224=1107.675,188.164,-66.178,-179.098,9.239,149.560
C05225=1107.679,187.915,-66.154,-179.099,9.236,149.560
C05226=1107.683,187.703,-66.132,-179.102,9.233,149.560
C05227=1107.686,187.490,-66.111,-179.104,9.231,149.560
C05228=1107.690,187.276,-66.090,-179.106,9.229,149.560
C05229=1107.694,187.063,-66.069,-179.108,9.226,149.560
C05230=1107.698,186.850,-66.049,-179.110,9.224,149.560
C05231=1107.702,186.637,-66.027,-179.111,9.222,149.560
C05232=1107.706,186.424,-66.007,-179.113,9.219,149.560
C05233=1107.710,186.211,-65.986,-179.115,9.217,149.560
C05234=1107.714,185.962,-65.962,-179.118,9.214,149.560
C05235=1107.719,185.714,-65.937,-179.120,9.211,149.559
C05236=1107.723,185.464,-65.913,-179.122,9.208,149.559
C05237=1107.728,185.216,-65.889,-179.125,9.205,149.559
C05238=1107.733,184.967,-65.864,-179.127,9.202,149.559
C05239=1107.736,184.718,-65.839,-179.129,9.200,149.559
C05240=1107.742,184.470,-65.815,-179.132,9.197,149.559
C05241=1107.746,184.221,-65.791,-179.134,9.194,149.559
C05242=1107.751,183.972,-65.767,-179.136,9.191,149.559
C05243=1107.754,183.723,-65.743,-179.139,9.188,149.559
C05244=1107.760,183.474,-65.718,-179.141,9.185,149.559
C05245=1107.764,183.226,-65.694,-179.143,9.183,149.559
C05246=1107.768,182.977,-65.670,-179.145,9.180,149.559
C05247=1107.773,182.728,-65.645,-179.148,9.177,149.559
C05248=1107.778,182.479,-65.622,-179.149,9.174,149.559
C05249=1107.782,182.231,-65.598,-179.152,9.171,149.559
C05250=1107.786,181.982,-65.574,-179.155,9.168,149.559
C05251=1107.791,181.733,-65.548,-179.157,9.164,149.559
C05252=1107.795,181.484,-65.524,-179.159,9.162,149.559
C05253=1107.800,181.235,-65.501,-179.161,9.159,149.559
C05254=1107.804,180.987,-65.477,-179.164,9.156,149.558
C05255=1107.810,180.738,-65.452,-179.166,9.154,149.558
C05256=1107.814,180.488,-65.429,-179.168,9.150,149.558
C05257=1107.818,180.240,-65.404,-179.170,9.147,149.558
C05258=1107.822,179.992,-65.380,-179.173,9.144,149.558
C05259=1107.827,179.743,-65.357,-179.176,9.141,149.558
C05260=1107.832,179.494,-65.333,-179.177,9.138,149.558
C05261=1107.836,179.245,-65.308,-179.180,9.135,149.558
C05262=1107.841,178.996,-65.285,-179.182,9.132,149.558
C05263=1107.845,178.747,-65.261,-179.184,9.130,149.558
C05264=1107.850,178.499,-65.236,-179.186,9.126,149.557
C05265=1107.854,178.250,-65.213,-179.189,9.123,149.557
C05266=1107.859,178.001,-65.189,-179.190,9.121,149.557
C05267=1107.863,177.752,-65.165,-179.193,9.117,149.557
C05268=1107.868,177.503,-65.141,-179.195,9.114,149.557
C05269=1107.872,177.255,-65.117,-179.197,9.112,149.557
C05270=1107.877,177.005,-65.093,-179.199,9.108,149.557
C05271=1107.881,176.757,-65.069,-179.202,9.105,149.557
C05272=1107.886,176.508,-65.046,-179.203,9.103,149.557
C05273=1107.890,176.260,-65.022,-179.206,9.099,149.556
C05274=1107.895,176.011,-64.998,-179.207,9.097,149.556
C05275=1107.899,175.761,-64.974,-179.210,9.094,149.556
C05276=1107.904,175.512,-64.951,-179.212,9.091,149.556
C05277=1107.908,175.264,-64.926,-179.214,9.088,149.556
C05278=1107.913,175.015,-64.903,-179.216,9.085,149.556
C05279=1107.917,174.766,-64.880,-179.219,9.082,149.556
C05280=1107.922,174.518,-64.856,-179.220,9.079,149.556
C05281=1107.927,174.269,-64.832,-179.223,9.076,149.556
C05282=1107.931,174.055,-64.811,-179.225,9.074,149.556
C05283=1107.935,173.842,-64.791,-179.226,9.071,149.555
C05284=1107.938,173.629,-64.771,-179.228,9.069,149.555
C05285=1107.942,173.416,-64.751,-179.231,9.066,149.555
C05286=1107.946,173.203,-64.731,-179.232,9.063,149.555
C05287=1107.950,172.989,-64.711,-179.234,9.060,149.555
C05288=1107.954,172.776,-64.690,-179.236,9.058,149.555
C05289=1107.958,172.563,-64.670,-179.238,9.056,149.555
C05290=1107.962,172.314,-64.646,-179.240,9.052,149.555
C05291=1107.967,172.065,-64.623,-179.242,9.050,149.555
C05292=1107.971,171.816,-64.599,-179.244,9.047,149.555
C05293=1107.976,171.568,-64.575,-179.246,9.043,149.554
C05294=1107.980,171.319,-64.552,-179.248,9.041,149.554
C05295=1107.985,171.070,-64.529,-179.251,9.038,149.554
C05296=1107.990,170.821,-64.505,-179.253,9.034,149.554
C05297=1107.994,170.572,-64.481,-179.255,9.032,149.554
C05298=1107.998,170.324,-64.458,-179.257,9.029,149.554
C05299=1108.003,170.074,-64.435,-179.259,9.026,149.554
C05300=1108.008,169.825,-64.412,-179.261,9.023,149.554
C05301=1108.012,169.576,-64.388,-179.263,9.020,149.554
C05302=1108.017,169.328,-64.364,-179.266,9.017,149.554
C05303=1108.021,169.079,-64.341,-179.268,9.014,149.554
C05304=1108.026,168.830,-64.318,-179.270,9.011,149.553
C05305=1108.031,168.581,-64.294,-179.272,9.008,149.553
C05306=1108.035,168.332,-64.271,-179.274,9.005,149.553
C05307=1108.040,168.084,-64.248,-179.276,9.002,149.553
C05308=1108.045,167.835,-64.225,-179.279,8.999,149.553
C05309=1108.049,167.586,-64.201,-179.280,8.996,149.553
C05310=1108.054,167.337,-64.178,-179.283,8.993,149.553
C05311=1108.058,167.089,-64.155,-179.285,8.990,149.553
C05312=1108.063,166.840,-64.132,-179.288,8.986,149.552
C05313=1108.067,166.591,-64.108,-179.289,8.984,149.552
C05314=1108.072,166.342,-64.085,-179.291,8.981,149.552
C05315=1108.077,166.093,-64.061,-179.294,8.977,149.552
C05316=1108.081,165.844,-64.039,-179.295,8.975,149.552
C05317=1108.085,165.595,-64.015,-179.298,8.972,149.552
C05318=1108.090,165.346,-63.992,-179.301,8.968,149.552
C05319=1108.095,165.097,-63.969,-179.302,8.966,149.552
C05320=1108.099,164.849,-63.946,-179.304,8.963,149.551
C05321=1108.104,164.600,-63.923,-179.307,8.959,149.551
C05322=1108.109,164.351,-63.899,-179.308,8.957,149.551
C05323=1108.113,164.102,-63.877,-179.311,8.953,149.551
C05324=1108.117,163.853,-63.853,-179.313,8.950,149.551
C05325=1108.122,163.604,-63.830,-179.315,8.947,149.551
C05326=1108.126,163.355,-63.808,-179.317,8.944,149.551
C05327=1108.132,163.106,-63.785,-179.319,8.941,149.550
C05328=1108.136,162.857,-63.762,-179.322,8.938,149.550
C05329=1108.140,162.608,-63.739,-179.323,8.935,149.550
C05330=1108.145,162.359,-63.715,-179.326,8.932,149.550
C05331=1108.150,162.110,-63.692,-179.328,8.929,149.550
C05332=1108.154,161.862,-63.669,-179.330,8.925,149.550
C05333=1108.159,161.613,-63.647,-179.332,8.923,149.550
C05334=1108.163,161.364,-63.624,-179.334,8.919,149.549
C05335=1108.168,161.115,-63.601,-179.336,8.916,149.549
C05336=1108.173,160.866,-63.578,-179.338,8.913,149.549
C05337=1108.177,160.617,-63.555,-179.340,8.910,149.549
C05338=1108.181,160.404,-63.535,-179.342,8.908,149.549
C05339=1108.185,160.191,-63.516,-179.344,8.904,149.549
C05340=1108.189,159.977,-63.496,-179.346,8.902,149.549
C05341=1108.193,159.764,-63.477,-179.348,8.899,149.548
C05342=1108.197,159.550,-63.457,-179.349,8.897,149.548
C05343=1108.201,159.337,-63.437,-179.351,8.894,149.548
C05344=1108.204,159.124,-63.419,-179.353,8.891,149.548
C05345=1108.208,158.911,-63.399,-179.355,8.889,149.548
C05346=1108.213,158.662,-63.376,-179.357,8.885,149.548
C05347=1108.217,158.413,-63.353,-179.358,8.882,149.547
C05348=1108.222,158.164,-63.330,-179.361,8.879,149.547
C05349=1108.226,157.915,-63.308,-179.363,8.876,149.547
C05350=1108.231,157.665,-63.285,-179.365,8.872,149.547
C05351=1108.236,157.417,-63.263,-179.368,8.869,149.547
C05352=1108.241,157.168,-63.239,-179.369,8.866,149.547
C05353=1108.245,156.919,-63.217,-179.371,8.863,149.546
C05354=1108.250,156.671,-63.194,-179.373,8.860,149.546
C05355=1108.254,156.421,-63.172,-179.376,8.856,149.546
C05356=1108.259,156.172,-63.149,-179.377,8.854,149.546
C05357=1108.263,155.924,-63.126,-179.379,8.850,149.546
C05358=1108.268,155.675,-63.104,-179.381,8.847,149.545
C05359=1108.273,155.426,-63.081,-179.384,8.844,149.545
C05360=1108.277,155.177,-63.059,-179.386,8.840,149.545
C05361=1108.282,154.928,-63.036,-179.387,8.837,149.545
C05362=1108.287,154.679,-63.014,-179.390,8.834,149.545
C05363=1108.291,154.430,-62.991,-179.392,8.830,149.545
C05364=1108.296,154.181,-62.969,-179.394,8.827,149.544
C05365=1108.300,153.932,-62.947,-179.396,8.824,149.544
C05366=1108.305,153.683,-62.923,-179.398,8.820,149.544
C05367=1108.310,153.434,-62.902,-179.400,8.818,149.544
C05368=1108.314,153.186,-62.879,-179.402,8.814,149.544
C05369=1108.319,152.936,-62.856,-179.404,8.811,149.543
C05370=1108.323,152.688,-62.834,-179.406,8.807,149.543
C05371=1108.328,152.439,-62.812,-179.408,8.804,149.543
C05372=1108.333,152.189,-62.789,-179.410,8.800,149.543
C05373=1108.337,151.941,-62.767,-179.412,8.798,149.543
C05374=1108.342,151.692,-62.745,-179.414,8.794,149.542
C05375=1108.347,151.443,-62.723,-179.416,8.791,149.542
C05376=1108.351,151.194,-62.700,-179.418,8.787,149.542
C05377=1108.355,150.945,-62.678,-179.420,8.784,149.542
C05378=1108.361,150.696,-62.655,-179.422,8.780,149.541
C05379=1108.365,150.447,-62.633,-179.425,8.777,149.541
C05380=1108.370,150.198,-62.611,-179.427,8.773,149.541
C05381=1108.374,149.949,-62.589,-179.428,8.771,149.541
C05382=1108.379,149.699,-62.566,-179.430,8.767,149.540
C05383=1108.384,149.451,-62.544,-179.432,8.763,149.540
C05384=1108.388,149.202,-62.522,-179.434,8.760,149.540
C05385=1108.393,148.953,-62.500,-179.436,8.756,149.539
C05386=1108.398,148.704,-62.478,-179.438,8.753,149.539
C05387=1108.403,148.455,-62.456,-179.440,8.749,149.539
C05388=1108.407,148.206,-62.433,-179.442,8.746,149.539
C05389=1108.412,147.958,-62.411,-179.444,8.742,149.539
C05390=1108.416,147.708,-62.389,-179.446,8.739,149.538
C05391=1108.421,147.459,-62.367,-179.448,8.735,149.538
C05392=1108.426,147.210,-62.345,-179.450,8.732,149.538
C05393=1108.430,146.961,-62.323,-179.452,8.729,149.537
C05394=1108.434,146.748,-62.304,-179.454,8.725,149.537
C05395=1108.438,146.535,-62.285,-179.455,8.723,149.537
C05396=1108.442,146.320,-62.266,-179.457,8.719,149.537
C05397=1108.446,146.108,-62.248,-179.459,8.717,149.536
C05398=1108.450,145.894,-62.228,-179.460,8.714,149.536
C05399=1108.454,145.681,-62.210,-179.462,8.710,149.536
C05400=1108.458,145.468,-62.191,-179.463,8.707,149.536
C05401=1108.462,145.254,-62.172,-179.465,8.704,149.535
C05402=1108.467,145.005,-62.151,-179.467,8.701,149.535
C05403=1108.471,144.756,-62.129,-179.468,8.697,149.535
C05404=1108.476,144.507,-62.107,-179.470,8.694,149.534
C05405=1108.480,144.258,-62.085,-179.472,8.690,149.534
C05406=1108.486,144.009,-62.063,-179.473,8.687,149.534
C05407=1108.490,143.760,-62.041,-179.475,8.683,149.533
C05408=1108.495,143.511,-62.019,-179.477,8.680,149.533
C05409=1108.499,143.262,-61.997,-179.479,8.676,149.533
C05410=1108.504,143.013,-61.975,-179.480,8.673,149.532
C05411=1108.508,142.764,-61.953,-179.482,8.670,149.532
C05412=1108.513,142.515,-61.931,-179.484,8.666,149.532
C05413=1108.518,142.266,-61.910,-179.486,8.662,149.531
C05414=1108.522,142.017,-61.888,-179.487,8.659,149.531
C05415=1108.527,141.768,-61.866,-179.489,8.656,149.531
C05416=1108.531,141.519,-61.844,-179.491,8.652,149.530
C05417=1108.536,141.270,-61.823,-179.492,8.649,149.530
C05418=1108.541,141.020,-61.801,-179.494,8.646,149.530
C05419=1108.546,140.772,-61.779,-179.496,8.642,149.529
C05420=1108.550,140.523,-61.758,-179.498,8.638,149.529
C05421=1108.554,140.274,-61.736,-179.499,8.636,149.529
C05422=1108.559,140.025,-61.714,-179.501,8.632,149.529
C05423=1108.563,139.775,-61.693,-179.503,8.628,149.528
C05424=1108.568,139.527,-61.671,-179.504,8.625,149.528
C05425=1108.573,139.278,-61.650,-179.506,8.622,149.528
C05426=1108.577,139.029,-61.628,-179.508,8.618,149.527
C05427=1108.583,138.780,-61.607,-179.510,8.614,149.527
C05428=1108.587,138.531,-61.585,-179.511,8.612,149.527
C05429=1108.592,138.282,-61.563,-179.513,8.608,149.527
C05430=1108.597,138.033,-61.541,-179.515,8.604,149.526
C05431=1108.601,137.783,-61.520,-179.517,8.601,149.526
C05432=1108.605,137.535,-61.499,-179.519,8.598,149.526
C05433=1108.610,137.286,-61.477,-179.520,8.594,149.525
C05434=1108.615,137.036,-61.456,-179.522,8.591,149.525
C05435=1108.620,136.787,-61.434,-179.524,8.588,149.525
C05436=1108.625,136.539,-61.413,-179.525,8.584,149.524
C05437=1108.629,136.289,-61.391,-179.527,8.581,149.524
C05438=1108.633,136.040,-61.370,-179.529,8.578,149.524
C05439=1108.638,135.792,-61.348,-179.531,8.574,149.523
C05440=1108.643,135.543,-61.327,-179.533,8.570,149.523
C05441=1108.648,135.293,-61.305,-179.534,8.568,149.523
C05442=1108.653,135.044,-61.284,-179.536,8.564,149.523
C05443=1108.657,134.796,-61.263,-179.538,8.560,149.522
C05444=1108.661,134.546,-61.241,-179.539,8.558,149.522
C05445=1108.666,134.297,-61.220,-179.541,8.554,149.522
C05446=1108.671,134.048,-61.199,-179.543,8.550,149.521
C05447=1108.676,133.799,-61.178,-179.544,8.548,149.521
C05448=1108.680,133.550,-61.156,-179.546,8.544,149.521
C05449=1108.685,133.301,-61.135,-179.548,8.541,149.521
C05450=1108.689,133.088,-61.117,-179.549,8.538,149.520
C05451=1108.694,132.874,-61.098,-179.551,8.535,149.520
C05452=1108.697,132.660,-61.080,-179.552,8.532,149.520
C05453=1108.701,132.447,-61.063,-179.554,8.529,149.519
C05454=1108.705,132.233,-61.044,-179.556,8.526,149.519
C05455=1108.709,132.020,-61.026,-179.557,8.523,149.519
C05456=1108.712,131.806,-61.008,-179.559,8.520,149.519
C05457=1108.717,131.593,-60.989,-179.560,8.518,149.519
C05458=1108.722,131.344,-60.969,-179.562,8.514,149.518
C05459=1108.726,131.095,-60.947,-179.563,8.511,149.518
C05460=1108.732,130.846,-60.926,-179.565,8.508,149.518
C05461=1108.735,130.596,-60.905,-179.567,8.504,149.517
C05462=1108.740,130.348,-60.884,-179.569,8.501,149.517
C05463=1108.746,130.098,-60.863,-179.570,8.498,149.517
C05464=1108.750,129.850,-60.842,-179.573,8.494,149.517
C05465=1108.755,129.601,-60.821,-179.575,8.491,149.516
C05466=1108.759,129.351,-60.799,-179.576,8.488,149.516
C05467=1108.764,129.102,-60.779,-179.578,8.484,149.516
C05468=1108.769,128.853,-60.757,-179.580,8.481,149.515
C05469=1108.774,128.604,-60.736,-179.581,8.478,149.515
C05470=1108.778,128.355,-60.716,-179.583,8.474,149.515
C05471=1108.783,128.107,-60.694,-179.585,8.470,149.515
C05472=1108.787,127.857,-60.673,-179.586,8.468,149.514
C05473=1108.792,127.608,-60.652,-179.588,8.464,149.514
C05474=1108.797,127.359,-60.632,-179.590,8.461,149.514
C05475=1108.802,127.110,-60.610,-179.591,8.458,149.513
C05476=1108.807,126.861,-60.589,-179.594,8.454,149.513
C05477=1108.811,126.612,-60.569,-179.596,8.451,149.513
C05478=1108.816,126.363,-60.548,-179.597,8.448,149.513
C05479=1108.821,126.114,-60.528,-179.599,8.444,149.512
C05480=1108.825,125.864,-60.506,-179.601,8.441,149.512
C05481=1108.829,125.615,-60.485,-179.602,8.438,149.512
C05482=1108.835,125.366,-60.464,-179.604,8.434,149.512
C05483=1108.839,125.117,-60.444,-179.606,8.430,149.511
C05484=1108.844,124.868,-60.423,-179.607,8.428,149.511
C05485=1108.849,124.619,-60.403,-179.609,8.424,149.511
C05486=1108.854,124.370,-60.382,-179.611,8.421,149.510
C05487=1108.858,124.121,-60.361,-179.613,8.417,149.510
C05488=1108.863,123.872,-60.340,-179.614,8.414,149.510
C05489=1108.867,123.622,-60.319,-179.617,8.411,149.510
C05490=1108.871,123.373,-60.299,-179.619,8.407,149.509
C05491=1108.877,123.124,-60.278,-179.620,8.404,149.509
C05492=1108.881,122.875,-60.257,-179.622,8.401,149.509
C05493=1108.886,122.626,-60.236,-179.624,8.397,149.508
C05494=1108.891,122.377,-60.216,-179.625,8.394,149.508
C05495=1108.896,122.128,-60.195,-179.627,8.390,149.508
C05496=1108.900,121.879,-60.175,-179.629,8.387,149.508
C05497=1108.905,121.630,-60.154,-179.630,8.384,149.507
C05498=1108.910,121.381,-60.133,-179.632,8.381,149.507
C05499=1108.914,121.132,-60.113,-179.634,8.377,149.507
C05500=1108.919,120.883,-60.092,-179.635,8.374,149.506
C05501=1108.924,120.633,-60.071,-179.637,8.371,149.506
C05502=1108.928,120.385,-60.051,-179.640,8.367,149.506
C05503=1108.934,120.135,-60.030,-179.641,8.363,149.506
C05504=1108.938,119.886,-60.010,-179.643,8.361,149.505
C05505=1108.942,119.637,-59.989,-179.645,8.357,149.505
